// TIA Portal project "СrystallizerGorodenki" (V14)

(* hardware
DEVICE "ET 200SP station_1"  ET 200SP-Station
   slot 0: "Rack_0"  Rack  6ES5 710-8MAx1
   slot 1: "PLC_1"  CPU 1510SP-1 PN  6ES7 510-1DJ01-0AB0  V2.1
   slot 2: "AI 4xRTD/TC 2-,3-,4-wire HF_1"  AI 4xRTD/TC 2-,3-,4-wire HF  6ES7 134-6JD00-0CA1  V2.0
      slot 1: "AI 4xRTD/TC 2-,3-,4-wire HF_1"  AI 4xRTD/TC 2-,3-,4-wire HF
   slot 3: "AI 4xRTD/TC 2-,3-,4-wire HF_2"  AI 4xRTD/TC 2-,3-,4-wire HF  6ES7 134-6JD00-0CA1  V2.0
      slot 1: "AI 4xRTD/TC 2-,3-,4-wire HF_2"  AI 4xRTD/TC 2-,3-,4-wire HF
   slot 4: "AI 4xRTD/TC 2-,3-,4-wire HF_3"  AI 4xRTD/TC 2-,3-,4-wire HF  6ES7 134-6JD00-0CA1  V2.0
      slot 1: "AI 4xRTD/TC 2-,3-,4-wire HF_3"  AI 4xRTD/TC 2-,3-,4-wire HF
   slot 5: "AI 4xI 2-,4-wire ST_1"  AI 4xI 2-,4-wire ST  6ES7 134-6GD00-0BA1  V1.1
      slot 1: "AI 4xI 2-,4-wire ST_1"  AI 4xI 2-,4-wire ST
   slot 6: "AI 4xI 2-,4-wire ST_2"  AI 4xI 2-,4-wire ST  6ES7 134-6GD00-0BA1  V1.1
      slot 1: "AI 4xI 2-,4-wire ST_2"  AI 4xI 2-,4-wire ST
   slot 7: "DI 16x24VDC ST_1"  DI 16x24VDC ST  6ES7 131-6BH01-0BA0  V0.0
      slot 1: "DI 16x24VDC ST_1"  DI 16x24VDC ST
   slot 8: "DI 16x24VDC ST_2"  DI 16x24VDC ST  6ES7 131-6BH01-0BA0  V0.0
      slot 1: "DI 16x24VDC ST_2"  DI 16x24VDC ST
   slot 9: "DI 16x24VDC ST_3"  DI 16x24VDC ST  6ES7 131-6BH01-0BA0  V0.0
      slot 1: "DI 16x24VDC ST_3"  DI 16x24VDC ST
   slot 10: "DI 8x24VDC ST_1"  DI 8x24VDC ST  6ES7 131-6BF01-0BA0  V0.0
      slot 1: "DI 8x24VDC ST_1"  DI 8x24VDC ST
   slot 11: "DQ 16x24VDC/0.5A ST_1"  DQ 16x24VDC/0.5A ST  6ES7 132-6BH01-0BA0  V0.0
      slot 1: "DQ 16x24VDC/0.5A ST_1"  DQ 16x24VDC/0.5A ST
   slot 12: "DQ 8x24VDC/0.5A ST_1"  DQ 8x24VDC/0.5A ST  6ES7 132-6BF01-0BA0  V0.0
      slot 1: "DQ 8x24VDC/0.5A ST_1"  DQ 8x24VDC/0.5A ST
   slot 13: "AQ 2xI ST_1"  AQ 2xI ST  6ES7 135-6GB00-0BA1  V1.0
      slot 1: "AQ 2xI ST_1"  AQ 2xI ST
   slot 14: "Server module_1"  Server module  6ES7 193-6PA00-0AA0  V1.1
      slot 1: "Server module_1"  Server module
   slot 127: "BA 2xRJ45"  BA 2xRJ45  6ES7 193-6AR00-0AA0  V0.0
      slot 32769: "Port_1"  6ES7 193-6AR00-0AA0
      slot 32770: "Port_2"  6ES7 193-6AR00-0AA0
DEVICE "HMI_1"  TP900 Comfort
   slot 0: "TP900 Comfort"  TP900 Comfort  6AV2 124-0JC01-0AX0  14.0.1.0
   slot 1: "HMI_RT_1"  TP900 Comfort  6AV2 124-0JC01-0AX0  14.0.1.0
   slot 5: "HMI_1.IE_CP_1"  PROFINET Interface  14.0.1.0
      slot 1: "PROFINET Interface_1"  PROFINET Interface
         slot 1: "Port_1"  Port
         slot 2: "Port_2"  Port
   slot 7: "HMI_1.MPI/DP_CP_1"  MPI/DP Interface  14.0.1.0
DEVICE "GSD device_1"  GSD.Device.PN
   slot 0: "Rack"  Rack  V1.0
   slot 0: "CTEU-PN"  CTEU-PN  2201471  V1.0.0
      slot 0: "CTEU-PN"  CTEU-PN
      slot 1: "PN-IO Interface"  PN-IO Interface
         slot 1: "Port 1"  Port 1
         slot 2: "Port 2"  Port 2
   slot 1: "VAEM-L1-S-16-PT_1"  VAEM-L1-S-16-PT  573939
      slot 0: "VAEM-L1-S-16-PT"  VAEM-L1-S-16-PT
DEVICE "SINAMICS G_1"  Sinamics.Device
   slot 0: "	_0"  Rail
   slot 0: "M1_1"  G120C PN  6SL3210-1KE18-8UF1  4.7.6
      slot 3: "PM G120C"  PM G120C  6SL3210-1KE18-8UF1  -
DEVICE "SINAMICS G_2"  Sinamics.Device
   slot 0: "	_0"  Rail
   slot 0: "M2_1"  G120C PN  6SL3210-1KE18-8UF1  4.7.6
      slot 3: "PM G120C"  PM G120C  6SL3210-1KE18-8UF1  -
DEVICE "SINAMICS G_4"  Sinamics.Device
   slot 0: "	_0"  Rail
   slot 0: "M7_1"  G120C PN  6SL3210-1KE18-8UF1  4.7.6
      slot 3: "PM G120C"  PM G120C  6SL3210-1KE18-8UF1  -
DEVICE "SINAMICS G_5"  Sinamics.Device
   slot 0: "	_0"  Rail
   slot 0: "M7_2"  G120C PN  6SL3210-1KE21-3UF1  4.7.6
      slot 3: "PM G120C"  PM G120C  6SL3210-1KE21-3UF1  -
DEVICE "PC-System_1"  SIMATIC PC station
   slot 0: "PC station"  Rail  SIMATIC PC-Station  V1.0
      slot 125: "Stationmanager"  Station_Manager  V6.0.4
   slot 1: "IE general_1"  IE General  IE_CP  V8.2.0
   slot 2: "HMI_RT_3"  WinCC RT Advanced  6AV2 104-0xxxx-xxxx  14.0.1.0
      slot 33792: "Host interface"  Host interface
*)

// ===== PLC "PLC_1"  CPU 1510SP-1 PN =====

VAR_GLOBAL   // PLC tag table "Default tag table"
   "Ai_TE1.1" AT %IW0 : Int;
   "Ai_TE1.2" AT %IW2 : Int;
   "Ai_TE1.3" AT %IW4 : Int;
   "Ai_TE2.1" AT %IW6 : Int;
   "Ai_TE2.2" AT %IW8 : Int;
   "Ai_TE2.3" AT %IW10 : Int;
   "Ai_TE7.1" AT %IW12 : Int;
   "Ai_TE7.2" AT %IW14 : Int;
   "Ai_TE3.1" AT %IW16 : Int;
   "Ai_TE3.2" AT %IW18 : Int;
   "Ai_TE3.3" AT %IW20 : Int;
   "Ai_LIC1.1" AT %IW24 : Int;
   "Ai_LIC2.1" AT %IW28 : Int;
   "Ai_LIC7.1" AT %IW32 : Int;
   "Ai_LIC7.2" AT %IW38 : Int;
   "Di_KF01" AT %I40.0 : Bool;
   "Di_AvarStop" AT %I40.1 : Bool;
   "Di_ACK" AT %I40.2 : Bool;
   "Di_BatRaz" AT %I40.3 : Bool;
   "Di_BatFault" AT %I40.4 : Bool;
   "Di_Bat24Ok" AT %I40.5 : Bool;
   "Di_BatEnable" AT %I40.6 : Bool;
   "Di_Qf1.1" AT %I40.7 : Bool;
   "Di_Km1.2" AT %I41.0 : Bool;
   "Di_Qf2.1" AT %I41.1 : Bool;
   "Di_Km2.2" AT %I41.2 : Bool;
   "Di_Qf3.1" AT %I41.3 : Bool;
   "Di_Km3.2" AT %I41.4 : Bool;
   "Di_Km03" AT %I42.0 : Bool;
   "Di_Km04" AT %I42.1 : Bool;
   "Di_QF7.1" AT %I42.2 : Bool;
   "Di_QF7.2" AT %I42.3 : Bool;
   "Di_Km10" AT %I42.4 : Bool;
   "Di_Ksp01" AT %I42.5 : Bool;
   "Di_Lah1.1" AT %I42.6 : Bool;
   "Di_Lah2.1" AT %I42.7 : Bool;
   "Di_Lah3.1" AT %I43.0 : Bool;
   "Di_Lah01" AT %I43.1 : Bool;
   "Di_Lal01" AT %I43.2 : Bool;
   "Di_Ga1.1" AT %I44.0 : Bool;
   "Di_Ga1.2" AT %I44.1 : Bool;
   "Di_Ga1.3" AT %I44.2 : Bool;
   "Di_Ga1.4" AT %I44.3 : Bool;
   "Di_Ga2.1" AT %I44.4 : Bool;
   "Di_Ga2.2" AT %I44.5 : Bool;
   "Di_Ga2.3" AT %I44.6 : Bool;
   "Di_Ga2.4" AT %I44.7 : Bool;
   "Di_Ga3.1" AT %I45.0 : Bool;
   "Di_Ga3.2" AT %I45.1 : Bool;
   "Di_Ga3.3" AT %I45.2 : Bool;
   "Di_Ga3.4" AT %I45.3 : Bool;
   "Di_Ga7.3" AT %I45.4 : Bool;
   "Di_Ga7.4" AT %I45.5 : Bool;
   "Di_1Ga01" AT %I45.6 : Bool;
   "Di_1Ga02" AT %I46.0 : Bool;
   "Di_1Ga03" AT %I46.1 : Bool;
   "Di_1Ga04" AT %I46.2 : Bool;
   "Di_1Ga05" AT %I46.3 : Bool;
   "Di_1Ga06" AT %I46.4 : Bool;
   "Di_Ga1.7" AT %I46.5 : Bool;
   "Di_Ga2.7" AT %I46.6 : Bool;
   "Di_Ga3.7" AT %I46.7 : Bool;
   "Dq_KB1" AT %Q0.0 : Bool;
   "Dq_Km1.2" AT %Q0.1 : Bool;
   "Dq_Km2.2" AT %Q0.2 : Bool;
   "Dq_Km3.2" AT %Q0.3 : Bool;
   "Dq_Km3" AT %Q0.4 : Bool;
   "Dq_Km4" AT %Q0.5 : Bool;
   "Dq_Km10" AT %Q0.6 : Bool;
   "Dq_V7.1" AT %Q0.7 : Bool;
   "Dq_V7.2" AT %Q1.0 : Bool;
   "Dq_V1.1" AT %Q3.0 : Bool;
   "Dq_V2.1" AT %Q3.1 : Bool;
   "Dq_V3.1" AT %Q3.2 : Bool;
   "Dq_V1.7" AT %Q3.3 : Bool;
   "Dq_V2.7" AT %Q3.4 : Bool;
   "Dq_V3.7" AT %Q3.5 : Bool;
   "Dq_V7.3" AT %Q3.6 : Bool;
   "Dq_V7.4" AT %Q3.7 : Bool;
   "System_Byte" AT %MB0 : Byte;
   "_Start" AT %M0.0 : Bool;   // Первый цикл
   "DiagStatusUpdate" AT %M0.1 : Bool;
   "_T(1)" AT %M0.2 : Bool;   // Всегда TRUE
   "_F(0)" AT %M0.3 : Bool;   // Всегда FALSE
   "_Clock" AT %MB1 : Byte;   // Байт часов
   "_Clk01sec" AT %M1.0 : Bool;   // Период изменения бита - 0.1 сек
   "_Clk02sec" AT %M1.1 : Bool;   // Период изменения бита - 0.2 сек
   "_Clk04sec" AT %M1.2 : Bool;   // Период изменения бита - 0.4 сек
   "_Clk05sec" AT %M1.3 : Bool;   // Период изменения бита - 0.5 сек
   "_Clk08sec" AT %M1.4 : Bool;   // Период изменения бита - 0.8 сек
   "_Clk10sec" AT %M1.5 : Bool;   // Период изменения бита - 1.0 сек
   "_Clk16sec" AT %M1.6 : Bool;   // Период изменения бита - 1.6 сек
   "_Clk20sec" AT %M1.7 : Bool;   // Период изменения бита - 2.0 сек
   "_ReStart" AT %M2.0 : Bool;   // Выполняется первый проход OB1
   "_AiMd" AT %M2.1 : Bool;   // Принудительная настройка аналоговых каналов
   "_HALT" AT %M2.2 : Bool;   // Общий "Аварийный СТОП"
   "_ACK" AT %M2.3 : Bool;   // Общий "Квитирование"
   "_MEn" AT %M2.4 : Bool;   // Общее разрешение сообщений
   "_Time" AT %MD20 : Time;   // Текущее системное время
   "_Time_dR" AT %MD24 : Real;   // Время цикла
   "Ao_RV01" AT %QW7 : Int;
   "Tag_3" AT %M11.0 : Bool;
   "Tag_4" AT %M11.1 : Bool;
   "Tag_5" AT %M11.2 : Bool;
   "Tag_6" AT %M11.3 : Bool;
END_VAR

VAR_GLOBAL CONSTANT   // PLC tag table "Default tag table"
   "NLoo" : Real := -1.0e+38;   // Условный уровень -oo для показаний датчика
   "NHoo" : Real := 1.0e+38;   // Условный уровень +oo для показаний датчика
   "TS0" : LDT := LDT#1970-01-01-00:00:00;   // Program_Alarm.TIMESTAMP := #TS0
   "Tz" : Time := T#0ms;   // Инициализация переменных времени
END_VAR

TYPE "PID"
   STRUCT
      Man_On : Bool;
      Man : Real;
      Sp : Real;
      LMN : Real;
   END_STRUCT;
END_TYPE

// folder: _LIB

TYPE "DrvST"
TITLE = 'Структура слова командного канала DrvCell побайтно'
VERSION : 0.1
   STRUCT
      STx : Byte := 16#00;   // [0_] Статус механизма
      WKx : Byte := 16#00;   // [1_] Вспомогательные данные канала
      Cmd : Byte := 16#00;   // [2_] Текущая команда и штамп идентификатора команды
      SPx : SInt := 0;   // [3_] Текущая уставка (-100..+100)[%]
   END_STRUCT;
END_TYPE

TYPE "DrvCF"
TITLE = 'Структура слова командного канала DrvCell побитно'
VERSION : 0.1
   STRUCT
      Sx1 : Bool := 0;   // [00] SQ канала Km1
      Sx2 : Bool := 0;   // [01] SQ канала Km2
      Ks1 : Bool := 0;   // [02] Включен канал Km1
      Ks2 : Bool := 0;   // [03] Включен канал Km2
      Tm1 : Bool := 0;   // [04] Время Tm1 истекло
      Tm2 : Bool := 0;   // [05] Время Tm2 истекло
      Er1 : Bool := 0;   // [06] Неисправность Km1
      Er2 : Bool := 0;   // [07] Неисправность Km2
      Act : Bool := 0;   // [10] Актуальность данных (контроль обрыва связи)
      Ack : Bool := 0;   // [11] Квитирование ошибок
      MsD : Bool := 0;   // [12] Сообщение: Наличие обрыва связи
      MsB : Bool := 0;   // [13] Сообщение: Наличие блокировки команды
      Mdx : Bool := 0;   // [14] Режим работы DrvCell (0==Ручной/1==Автомат)
      F15 : Bool := 0;   // [15] Резерв
      F16 : Bool := 0;   // [16] Резерв
      F17 : Bool := 0;   // [17] Резерв
      Cm0 : Bool := 0;   // [20] Команда: бит 0
      Cm1 : Bool := 0;   // [21] Команда: бит 1
      Cm2 : Bool := 0;   // [22] Команда: бит 2
      F23 : Bool := 0;   // [23] Резерв
      F24 : Bool := 0;   // [24] Резерв
      F25 : Bool := 0;   // [25] Резерв
      F26 : Bool := 0;   // [26] Резерв
      F27 : Bool := 0;   // [27] Резерв
      SPx : SInt := 0;   // [3_] Текущая уставка (-100..+100)[%]
   END_STRUCT;
END_TYPE

TYPE "DrvNm"
TITLE = 'Данные канала системы блокировок'
VERSION : 0.1
   STRUCT
      Ds1 : Bool := 0;   // Блокировка включения (принудительное отключение) Km1
      Ds2 : Bool := 0;   // Блокировка включения (принудительное отключение) Km2
      DsA : Bool := 0;   // Общая блокировка включения (принудительное отключение) Km1&Km2
      r03 : Bool := 0;   // ----
      r04 : Bool := 0;   // ----
      r05 : Bool := 0;   // ----
      r06 : Bool := 0;   // ----
      r07 : Bool := 0;   // ----
      MsA : Byte := 16#00;   // Номер сообщения общей блокировки
      Ms2 : Byte := 16#00;   // Номер сообщения блокировки включения Km2
      Ms1 : Byte := 16#00;   // Номер сообщения блокировки включения Km1
   END_STRUCT;
END_TYPE

TYPE "DrvMs"
TITLE = 'Расшифровка слова состояния HMI DrvCell побитно'
VERSION : 0.1
   STRUCT
      Ds1 : Bool := 0;   // Действие Km1 заблокировано (Ds1/DsA)
      Ds2 : Bool := 0;   // Действие Km2 заблокировано (Ds2/DsA)
      QFe : Bool := 0;   // Отключен автоматический выключатель
      Flt : Bool := 0;   // Внешняя неисправность (блокирующая)
      Err : Bool := 0;   // Внутренняя неисправность DrvCell
      b29 : Bool := 0;   // ----
      b30 : Bool := 0;   // ----
      b31 : Bool := 0;   // ----
      Sr1 : Bool := 0;   // Не сработал КВ SQ1 за заданное время Tm1
      Sr2 : Bool := 0;   // Не сработал КВ SQ2 за заданное время Tm2
      Se1 : Bool := 0;   // Механиз без команды сошел с КВ SQ1
      Se2 : Bool := 0;   // Механиз без команды сошел с КВ SQ2
      SeA : Bool := 0;   // Одновременно активны оба КВ SQ1 и SQ2
      KeB : Bool := 0;   // БК KxB не соответствует состоянию KOn
      Ke1 : Bool := 0;   // БК Kx1 не соответствует контактору Km1
      Ke2 : Bool := 0;   // БК Kx2 не соответствует контактору Km2
      Mdx : Bool := 0;   // Режим работы DrvCell (0==Ручной/1==Автомат)
      Lg2 : Bool := 0;   // Индикация действия от SB2 (зеленый)
      Ly2 : Bool := 0;   // Индикация действия от SB2 (желтый)
      Lr2 : Bool := 0;   // Индикация действия от SB2 (красный)
      HSB : Bool := 0;   // Доп. признак индикации SB2
      Lg1 : Bool := 0;   // Индикация действия от SB1 (зеленый)
      Ly1 : Bool := 0;   // Индикация действия от SB1 (желтый)
      Lr1 : Bool := 0;   // Индикация действия от SB1 (красный)
      Sx1 : Bool := 0;   // Активное состояние SQ1
      Sx2 : Bool := 0;   // Активное состояние SQ2
      Ks1 : Bool := 0;   // Запрос на включение Km1
      Ks2 : Bool := 0;   // Запрос на включение Km2
      Tm1 : Bool := 0;   // Время Tm1 истекло
      Tm2 : Bool := 0;   // Время Tm2 истекло
      Er1 : Bool := 0;   // Неисправность Km1
      Er2 : Bool := 0;   // Неисправность Km2
   END_STRUCT;
END_TYPE

TYPE "TPTR"
TITLE = 'Формат данных типа POINTER'
VERSION : 0.1
   STRUCT
      DN : UInt := 0;   // DB number
      AR : UDInt := 0;   // Memory area
   END_STRUCT;
END_TYPE

TYPE "TANY"
TITLE = 'Формат данных типа ANY'
VERSION : 0.1
   STRUCT
      S7 : Byte := B#16#00;   // 10h for S7
      TP : Byte := B#16#00;   // Data type
      RF : UInt := 0;   // Repetition factor
      PTR : "TPTR";   // POINTER
   END_STRUCT;
END_TYPE

TYPE "AiSP"
TITLE = 'Параметры настройки входного аналогового канала'
VERSION : 0.1
   STRUCT
      "M" : Struct   // Общая мастер-структура параметров каналов
         Rz : Bool := 1;   // При Rz<>Rs производится перерасчет канала
         Rs : Bool := 0;   // По фронту изменения Rs производится перенастройка канала
         Nm : Bool := 0;   // Pn указывает нормальный==0/номинальный==1 сигнал
         Ke : Bool := 0;   // Прямое использование Kf и Zp (с перерассчетом P1 и P0)
         Ms : Bool := 1;   // Разрешена генерация сообщений и использование Pn
         Rt : Bool := 0;   // Круговой датчик с переходом через 0 (однооборотный/многооборотный)
         Rh : Bool := 1;   // Для кругового датчика использовать шкалу со знаком (-180*..+180*)
         R0 : Word := 16#0000;   // ----
         An : DInt := DINT#27648;   // Значение PIW/PID(Ai/Ad) при 100% входного диапазона
         P1 : Real := 100.0;   // Номинал Px при Ai=100% (Ai=An[1]) [E]
         P0 : Real := 0.0;   // Номинал Px при Ai=0% (Ai=0[1]) [E]
         Kf : Real := 1.0;   // Коэффициент преобразования Ai=>Px (множитель) [E/1]
         Kx : Real := 1.0;   // Множитель для сглаживания колебаний входного сигнала
         dP : Real := 0.0;   // Гистерезис в определении уровней
      END_STRUCT;
      Pn : Real := 1.0e+38;   // Номинальный/Нормальный уровень сигнала [E]
      Ha : Real := 1.0e+38;   // Верхний уровень сигнала: Аварийный [E/%]
      La : Real := -1.0e+38;   // Нижний уровень сигнала: Аварийный [E/%]
      Hw : Real := 1.0e+38;   // Верхний уровень сигнала: Предупредительный [E/%]
      Lw : Real := -1.0e+38;   // Нижний уровень сигнала: Предупредительный [E/%]
      H1 : Real := 1.0e+38;   // Верхний уровень сигнала: Рабочая зона 1 [E/%]
      L1 : Real := -1.0e+38;   // Нижний уровень сигнала: Рабочая зона 1 [E/%]
      H0 : Real := 1.0e+38;   // Верхний уровень сигнала: Рабочая зона 0 [E/%]
      L0 : Real := -1.0e+38;   // Нижний уровень сигнала: Рабочая зона 0 [E/%]
   END_STRUCT;
END_TYPE

TYPE "DrvRd"
TITLE = 'Данные канала резервирования приводов'
VERSION : 0.1
   STRUCT
      S : Struct
         Mst : Bool := 1;   // Данный привод является основным (Master==1/Slave==0)
         Rd1 : Bool := 1;   // Данный привод включен как основной
         Rd2 : Bool := 0;   // Данный привод включен как резервный
         Dis : Bool := 0;   // Запрет использования привода (блокировка)
         r0 : Word := 16#0000;   // ---- Структура статуса (состояния) резерва
      END_STRUCT;
      "M" : Struct
         UBr : Bool := 0;   // Безусловное растормаживание (расжать)
         Enb : Bool := 0;   // Разрешение работы (разблокирование)
         KOn : Bool := 0;   // Включить намагничивание V=0 (команда)
         Run : Bool := 0;   // Пуск привода V=Vs (команда)
         Ack : Bool := 0;   // Сброс индикации ошибки (квитирование) (1==активен)
         Id : Word := 16#0000;   // Идентификатор дополнительных параметров привода
         Ms : Real := 0.0;   // Заданный момент [%]
         Vs : Real := 0.0;   // Заданная скорость [E]
         Vn : Real := 100.0;   // Номинальная скорость [E] Структура параметров мастера резерва
      END_STRUCT;
      X : Struct
         Brk : Bool := 0;   // Привод включен (разблокировка тормоза).
         Err : Bool := 0;   // Неисправность/авария привода
         Rdy : Bool := 0;   // Готовность привода к включению
         SW : Word := 16#0000;   // Текущее слово состояния привода
         Vx : Real := 0.0;   // Текущая скорость привода [E]
         Ix : Real := 0.0;   // Текущий ток привода [%]
         Mx : Real := 0.0;   // Текущий момент привода [%]
         An : Int := 0;   // Текущий номер сигнала Alarm [№] (предупреждение) (либо альтернативные данные)
         Fn : Int := 0;   // Текущий номер сигнала Fault [№] (отказ) Структура состояния привода
      END_STRUCT;
   END_STRUCT;
END_TYPE

TYPE "DrvME"
VERSION : 0.1
   STRUCT
      Pr : Struct   // Структура параметров сообщения ALARM
         N1 : UDInt := 0;   // Именная строка сообщения (MSGS=GRP)
         N2 : UDInt := 0;   // Признаки состояния сообщения (MSGS=MEn/Mdx/KOn)
         N3 : UDInt := 0;   // Основное сообщение (MSGS=A)
         N4 : UDInt := 0;   // Вспомогательное сообщение (MSGS=B)
         N5 : UDInt := 0;   // Вспомогательное сообщение (MSGS=C)
         N6 : UDInt := 0;   // Дополнительная строка сообщения (MSGS=GRP+N)
      END_STRUCT;
   END_STRUCT;
END_TYPE

TYPE "AiSF"
VERSION : 0.1
   STRUCT
      b24 : Bool;   // ----
      b25 : Bool;   // ----
      b26 : Bool;   // ----
      b27 : Bool;   // ----
      MEn : Bool;   // Разрешение выдачи сообщений (HMI)
      b29 : Bool;   // ----
      b30 : Bool;   // ----
      QSt : Bool;   // Настройка блока выполнена
      LSP : Bool;   // Запрос установки смещения (PLC)
      HSP : Bool;   // Запрос установки смещения (HMI)
      ESP : Bool;   // Разрешение установки смещения (HMI)
      QSP : Bool;   // Признак установки смещения
      LFQ : Bool;   // Запрос режима форсирования (PLC)
      HFQ : Bool;   // Запрос режима форсирования (HMI)
      EFQ : Bool;   // Разрешение режима форсирования (HMI)
      QFQ : Bool;   // Признак режима форсирования
      QWg : Bool;   // Наличие предупреждения
      QAm : Bool;   // Наличие аварии
      QFt : Bool;   // Наличие неисправности канала
      b11 : Bool;   // ----
      b12 : Bool;   // ----
      b13 : Bool;   // ----
      HWg : Bool;   // Наличие предупреждения (HMI:Yellow)
      HAm : Bool;   // Наличие аварии/неисправности (HMI:Red)
      QL0 : Bool;   // Нижний уровень сигнала: Рабочая зона 0
      QH0 : Bool;   // Верхний уровень сигнала: Рабочая зона 0
      QL1 : Bool;   // Нижний уровень сигнала: Рабочая зона 1
      QH1 : Bool;   // Верхний уровень сигнала: Рабочая зона 1
      QLw : Bool;   // Нижний уровень сигнала: Предупредительный
      QHw : Bool;   // Верхний уровень сигнала: Предупредительный
      QLa : Bool;   // Нижний уровень сигнала: Аварийный
      QHa : Bool;   // Верхний уровень сигнала: Аварийный
   END_STRUCT;
END_TYPE

// folder: Ai

DATA_BLOCK "AiCh_TE1.1"   // DB1
{ S7_Optimized_Access := 'FALSE' }
VERSION : 0.1
// stored: InstanceOfName AiCh_My
"AiCh_My"
BEGIN
END_DATA_BLOCK

DATA_BLOCK "AiCh_TE1.2"   // DB2
{ S7_Optimized_Access := 'FALSE' }
VERSION : 0.1
// stored: InstanceOfName AiCh_My
"AiCh_My"
BEGIN
END_DATA_BLOCK

DATA_BLOCK "AiCh_TE1.3"   // DB3
{ S7_Optimized_Access := 'FALSE' }
VERSION : 0.1
// stored: InstanceOfName AiCh_My
"AiCh_My"
BEGIN
END_DATA_BLOCK

DATA_BLOCK "AiCh_TE2.1"   // DB4
{ S7_Optimized_Access := 'FALSE' }
VERSION : 0.1
// stored: InstanceOfName AiCh_My
"AiCh_My"
BEGIN
END_DATA_BLOCK

DATA_BLOCK "AiCh_TE2.2"   // DB5
{ S7_Optimized_Access := 'FALSE' }
VERSION : 0.1
// stored: InstanceOfName AiCh_My
"AiCh_My"
BEGIN
END_DATA_BLOCK

DATA_BLOCK "AiCh_TE2.3"   // DB6
{ S7_Optimized_Access := 'FALSE' }
VERSION : 0.1
// stored: InstanceOfName AiCh_My
"AiCh_My"
BEGIN
END_DATA_BLOCK

DATA_BLOCK "AiCh_TE7.1"   // DB7
{ S7_Optimized_Access := 'FALSE' }
VERSION : 0.1
// stored: InstanceOfName AiCh_My
"AiCh_My"
BEGIN
END_DATA_BLOCK

DATA_BLOCK "AiCh_TE7.2"   // DB8
{ S7_Optimized_Access := 'FALSE' }
VERSION : 0.1
// stored: InstanceOfName AiCh_My
"AiCh_My"
BEGIN
END_DATA_BLOCK

DATA_BLOCK "AiCh_TE3.1"   // DB9
{ S7_Optimized_Access := 'FALSE' }
VERSION : 0.1
// stored: InstanceOfName AiCh_My
"AiCh_My"
BEGIN
END_DATA_BLOCK

DATA_BLOCK "AiCh_TE3.2"   // DB10
{ S7_Optimized_Access := 'FALSE' }
VERSION : 0.1
// stored: InstanceOfName AiCh_My
"AiCh_My"
BEGIN
END_DATA_BLOCK

DATA_BLOCK "AiCh_TE3.3"   // DB11
{ S7_Optimized_Access := 'FALSE' }
VERSION : 0.1
// stored: InstanceOfName AiCh_My
"AiCh_My"
BEGIN
END_DATA_BLOCK

DATA_BLOCK "AiCh_LIC1.1"   // DB12
{ S7_Optimized_Access := 'FALSE' }
VERSION : 0.1
// stored: InstanceOfName AiCh_My
"AiCh_My"
BEGIN
END_DATA_BLOCK

DATA_BLOCK "AiCh_LIC2.1"   // DB13
{ S7_Optimized_Access := 'FALSE' }
VERSION : 0.1
// stored: InstanceOfName AiCh_My
"AiCh_My"
BEGIN
END_DATA_BLOCK

DATA_BLOCK "AiCh_LIC3.1"   // DB14
{ S7_Optimized_Access := 'FALSE' }
VERSION : 0.1
// stored: InstanceOfName AiCh_My
"AiCh_My"
BEGIN
END_DATA_BLOCK

DATA_BLOCK "AiCh_LIC7.1"   // DB15
{ S7_Optimized_Access := 'FALSE' }
VERSION : 0.1
// stored: InstanceOfName AiCh_My
"AiCh_My"
BEGIN
END_DATA_BLOCK

DATA_BLOCK "AiCh_LIC7.2"   // DB16
{ S7_Optimized_Access := 'FALSE' }
VERSION : 0.1
// stored: InstanceOfName AiCh_My
"AiCh_My"
BEGIN
END_DATA_BLOCK

DATA_BLOCK "ForVO_DB"   // DB60
{ S7_Optimized_Access := 'FALSE' }
VERSION : 0.1
// stored: InstanceOfName ForVO
"ForVO"
BEGIN
END_DATA_BLOCK

// folder: Drives

DATA_BLOCK "DriveM1_1"   // DB33
{ S7_Optimized_Access := 'FALSE' }
AUTHOR : AA
FAMILY : xDEVICE
VERSION : 0.1
// stored: InstanceOfName MM_T352
"MM_T352"
BEGIN
END_DATA_BLOCK

DATA_BLOCK "DriveM7_1"   // DB34
{ S7_Optimized_Access := 'FALSE' }
AUTHOR : AA
FAMILY : xDEVICE
VERSION : 0.1
// stored: InstanceOfName MM_T352
"MM_T352"
BEGIN
END_DATA_BLOCK

DATA_BLOCK "DriveM7_2"   // DB35
{ S7_Optimized_Access := 'FALSE' }
AUTHOR : AA
FAMILY : xDEVICE
VERSION : 0.1
// stored: InstanceOfName MM_T352
"MM_T352"
BEGIN
END_DATA_BLOCK

DATA_BLOCK "DriveM2_1"   // DB38
{ S7_Optimized_Access := 'FALSE' }
AUTHOR : AA
FAMILY : xDEVICE
VERSION : 0.1
// stored: InstanceOfName MM_T352
"MM_T352"
BEGIN
END_DATA_BLOCK

// folder: Errors

DATA_BLOCK "FpDW_DB"   // DB43
{ S7_Optimized_Access := 'FALSE' }
VERSION : 0.1
// stored: InstanceOfName FpDW
"FpDW"
BEGIN
END_DATA_BLOCK

// folder: IceWater

DATA_BLOCK "IceWaterWork_DB"   // DB61
{ S7_Optimized_Access := 'TRUE' }
VERSION : 0.1
// stored: InstanceOfName IceWaterWork
"IceWaterWork"
BEGIN
END_DATA_BLOCK

// folder: KristalizersWork

DATA_BLOCK "Kr_2_Work"   // DB45
{ S7_Optimized_Access := 'TRUE' }
VERSION : 0.1
// stored: InstanceOfName KristalizerWork
"KristalizerWork"
BEGIN
END_DATA_BLOCK

DATA_BLOCK "Mixer2_Work_DB"   // DB47
{ S7_Optimized_Access := 'TRUE' }
VERSION : 0.1
// stored: InstanceOfName MixerWork
"MixerWork"
BEGIN
END_DATA_BLOCK

DATA_BLOCK "Mixer1_Work_DB"   // DB48
{ S7_Optimized_Access := 'TRUE' }
VERSION : 0.1
// stored: InstanceOfName MixerWork
"MixerWork"
BEGIN
END_DATA_BLOCK

DATA_BLOCK "Kr_1_Work"   // DB63
{ S7_Optimized_Access := 'TRUE' }
VERSION : 0.1
// stored: InstanceOfName KristalizerWork
"KristalizerWork"
BEGIN
END_DATA_BLOCK

// folder: Lines

DATA_BLOCK "ViewLine_DB"   // DB58
{ S7_Optimized_Access := 'TRUE' }
VERSION : 0.1
// stored: InstanceOfName ViewLine
"ViewLine"
BEGIN
END_DATA_BLOCK

// folder: Messages

DATA_BLOCK "Messages"   // DB44
{ S7_Optimized_Access := 'FALSE' }
VERSION : 0.1
   VAR
      Message1 : Bool;
      Message2 : Bool;
      Message3 : Bool;
      Message4 : Bool;
      Message5 : Bool;
      Message6 : Bool;
      Message7 : Bool;
      Message8 : Bool;
      Message9 : Bool;
      Message10 : Bool;
      Message11 : Bool;
      Message12 : Bool;
      Message13 : Bool;
      Message14 : Bool;
      Message15 : Bool;
      Message16 : Bool;
   END_VAR
BEGIN
END_DATA_BLOCK

// folder: Pumps&Valves

DATA_BLOCK "DrvCell_M1_2"   // DB17
{ S7_Optimized_Access := 'FALSE' }
AUTHOR : SAA
FAMILY : xDRIVER
NAME : DrvCell
VERSION : 4.0
// stored: InstanceOfName DrvCell
"DrvCell"
BEGIN
END_DATA_BLOCK

DATA_BLOCK "DrvCell_M2_2"   // DB18
{ S7_Optimized_Access := 'FALSE' }
AUTHOR : SAA
FAMILY : xDRIVER
NAME : DrvCell
VERSION : 4.0
// stored: InstanceOfName DrvCell
"DrvCell"
BEGIN
END_DATA_BLOCK

DATA_BLOCK "DrvCell_M3_2"   // DB19
{ S7_Optimized_Access := 'FALSE' }
AUTHOR : SAA
FAMILY : xDRIVER
NAME : DrvCell
VERSION : 4.0
// stored: InstanceOfName DrvCell
"DrvCell"
BEGIN
END_DATA_BLOCK

DATA_BLOCK "DrvCell_M3"   // DB20
{ S7_Optimized_Access := 'FALSE' }
AUTHOR : SAA
FAMILY : xDRIVER
NAME : DrvCell
VERSION : 4.0
// stored: InstanceOfName DrvCell
"DrvCell"
BEGIN
END_DATA_BLOCK

DATA_BLOCK "DrvCell_M4"   // DB21
{ S7_Optimized_Access := 'FALSE' }
AUTHOR : SAA
FAMILY : xDRIVER
NAME : DrvCell
VERSION : 4.0
// stored: InstanceOfName DrvCell
"DrvCell"
BEGIN
END_DATA_BLOCK

DATA_BLOCK "DrvCell_M10"   // DB22
{ S7_Optimized_Access := 'FALSE' }
AUTHOR : SAA
FAMILY : xDRIVER
NAME : DrvCell
VERSION : 4.0
// stored: InstanceOfName DrvCell
"DrvCell"
BEGIN
END_DATA_BLOCK

DATA_BLOCK "DrvCell_V7_1"   // DB23
{ S7_Optimized_Access := 'FALSE' }
AUTHOR : SAA
FAMILY : xDRIVER
NAME : DrvCell
VERSION : 4.0
// stored: InstanceOfName DrvCell
"DrvCell"
BEGIN
END_DATA_BLOCK

DATA_BLOCK "DrvCell_V7_2"   // DB24
{ S7_Optimized_Access := 'FALSE' }
AUTHOR : SAA
FAMILY : xDRIVER
NAME : DrvCell
VERSION : 4.0
// stored: InstanceOfName DrvCell
"DrvCell"
BEGIN
END_DATA_BLOCK

DATA_BLOCK "DrvCell_V1_1"   // DB25
{ S7_Optimized_Access := 'FALSE' }
AUTHOR : SAA
FAMILY : xDRIVER
NAME : DrvCell
VERSION : 4.0
// stored: InstanceOfName DrvCell
"DrvCell"
BEGIN
END_DATA_BLOCK

DATA_BLOCK "DrvCell_V2_1"   // DB26
{ S7_Optimized_Access := 'FALSE' }
AUTHOR : SAA
FAMILY : xDRIVER
NAME : DrvCell
VERSION : 4.0
// stored: InstanceOfName DrvCell
"DrvCell"
BEGIN
END_DATA_BLOCK

DATA_BLOCK "DrvCell_V3_1"   // DB27
{ S7_Optimized_Access := 'FALSE' }
AUTHOR : SAA
FAMILY : xDRIVER
NAME : DrvCell
VERSION : 4.0
// stored: InstanceOfName DrvCell
"DrvCell"
BEGIN
END_DATA_BLOCK

DATA_BLOCK "DrvCell_V1_7"   // DB28
{ S7_Optimized_Access := 'FALSE' }
AUTHOR : SAA
FAMILY : xDRIVER
NAME : DrvCell
VERSION : 4.0
// stored: InstanceOfName DrvCell
"DrvCell"
BEGIN
END_DATA_BLOCK

DATA_BLOCK "DrvCell_V2_7"   // DB29
{ S7_Optimized_Access := 'FALSE' }
AUTHOR : SAA
FAMILY : xDRIVER
NAME : DrvCell
VERSION : 4.0
// stored: InstanceOfName DrvCell
"DrvCell"
BEGIN
END_DATA_BLOCK

DATA_BLOCK "DrvCell_V3_7"   // DB30
{ S7_Optimized_Access := 'FALSE' }
AUTHOR : SAA
FAMILY : xDRIVER
NAME : DrvCell
VERSION : 4.0
// stored: InstanceOfName DrvCell
"DrvCell"
BEGIN
END_DATA_BLOCK

DATA_BLOCK "DrvCell_V7_3"   // DB31
{ S7_Optimized_Access := 'FALSE' }
AUTHOR : SAA
FAMILY : xDRIVER
NAME : DrvCell
VERSION : 4.0
// stored: InstanceOfName DrvCell
"DrvCell"
BEGIN
END_DATA_BLOCK

DATA_BLOCK "DrvCell_V7_4"   // DB32
{ S7_Optimized_Access := 'FALSE' }
AUTHOR : SAA
FAMILY : xDRIVER
NAME : DrvCell
VERSION : 4.0
// stored: InstanceOfName DrvCell
"DrvCell"
BEGIN
END_DATA_BLOCK

DATA_BLOCK "DrvCell_M1_1"   // DB36
{ S7_Optimized_Access := 'FALSE' }
AUTHOR : SAA
FAMILY : xDRIVER
NAME : DrvCell
VERSION : 4.0
// stored: InstanceOfName DrvCell
"DrvCell"
BEGIN
END_DATA_BLOCK

DATA_BLOCK "DrvCell_M2_1"   // DB37
{ S7_Optimized_Access := 'FALSE' }
AUTHOR : SAA
FAMILY : xDRIVER
NAME : DrvCell
VERSION : 4.0
// stored: InstanceOfName DrvCell
"DrvCell"
BEGIN
END_DATA_BLOCK

DATA_BLOCK "DrvCell_M7_1"   // DB39
{ S7_Optimized_Access := 'FALSE' }
AUTHOR : SAA
FAMILY : xDRIVER
NAME : DrvCell
VERSION : 4.0
// stored: InstanceOfName DrvCell
"DrvCell"
BEGIN
END_DATA_BLOCK

DATA_BLOCK "DrvCell_M7_2"   // DB40
{ S7_Optimized_Access := 'FALSE' }
AUTHOR : SAA
FAMILY : xDRIVER
NAME : DrvCell
VERSION : 4.0
// stored: InstanceOfName DrvCell
"DrvCell"
BEGIN
END_DATA_BLOCK

DATA_BLOCK "DrvCell_M5"   // DB59
{ S7_Optimized_Access := 'FALSE' }
AUTHOR : SAA
FAMILY : xDRIVER
NAME : DrvCell
VERSION : 4.0
// stored: InstanceOfName DrvCell
"DrvCell"
BEGIN
END_DATA_BLOCK

// folder: Share

DATA_BLOCK "Data"   // DB41
{ S7_Optimized_Access := 'TRUE' }
VERSION : 0.1
   VAR
      Ack : Bool;
      GlobalError : Bool;
      GlobalErrorStop : Bool;
   END_VAR
   VAR RETAIN
      Reg_01RV01 : "PID";
      Reg_M7_1 : "PID";
   END_VAR
   VAR
      Reg_M7_2 : "PID";
      Reg_TE1_1 : Struct
         In : Bool := FALSE;
         Sp : Real := 0.0;
         Gis : Real := 0.1;
         V1_1 : Bool := FALSE;
      END_STRUCT;
      Reg_TE2_1 : Struct
         In : Bool := FALSE;
         Sp : Real := 0.0;
         Gis : Real := 0.1;
         V2_1 : Bool := FALSE;
      END_STRUCT;
   END_VAR
   VAR RETAIN
      Mixer1 : Struct
         Man : Real;
         Start : Bool;
         Stop : Bool;
         RegimBothSide : Bool := true;
         Power : Real := 50.0;
         TimeRight : DInt := 60;
         TimeLeft : DInt := 60;
         TimePause : DInt := 60;
         Direction : Int;
      END_STRUCT;
      Mixer2 : Struct
         Man : Real;
         Start : Bool;
         Stop : Bool;
         RegimBothSide : Bool := true;
         Power : Real := 50.0;
         TimeRight : DInt := 60;
         TimeLeft : DInt := 60;
         TimePause : DInt := 60;
         Direction : Int;
      END_STRUCT;
   END_VAR
   VAR
      MAN_ON : Bool;
      washing : Struct
         cipRegim : Int := 1;
         readyGlobal : Bool;
         readyRoute : Bool;
         Start : Bool;
         Stop : Bool;
      END_STRUCT;
      LevelVO_Pv : Real;
   END_VAR
   VAR RETAIN
      TempIn_Sp : Real := 30.0;
      Power_7_2 : Real := 40.0;
      Power_7_2_CIP : Real := 40.0;
   END_VAR
   VAR
      Kr1 : Struct
         Regim : Int := 1;
         TempFilling : Real := 30.0;
         TempKristal : Real := 15.0;
         TimeKristal : Int := 8;
         Start : Bool;
         Stop : Bool;
         Ready_Route : Bool;
         Ready_Work : Bool;
         Kr1 : Struct
            Regim : Int := 1;
            TempFilling : Real := 30.0;
            TempKristal : Real := 15.0;
            TimeKristal : Int := 8;
            Start : Bool;
            Stop : Bool;
            Ready_Route : Bool;
            Ready_Work : Bool;
         END_STRUCT;
      END_STRUCT;
      Kr2 : Struct
         Regim : Int := 1;
         TempFilling : Real := 30.0;
         TempKristal : Real := 15.0;
         TimeKristal : Int := 8;
         Start : Bool;
         Stop : Bool;
         Ready_Route : Bool;
         Ready_Work : Bool;
      END_STRUCT;
      TE1_1_SP : Real;
      Mixer1_Run : Bool;
      Mixer2_Run : Bool;
      Front_Mixer_1 : Bool;
      Front_Mixer_2 : Bool;
      Erorrs_Beep : Bool;
      KR1_Beep : Bool;
      KR2_Beep : Bool;
      Equipment_Work : Bool;
      ReadyCIP : Bool;
      ReadyKr1 : Bool;
      ReadyKr2 : Bool;
   END_VAR
   VAR RETAIN
      EnableReady : Bool := true;
   END_VAR
BEGIN
   Reg_M7_1.Sp := 10.0;
   Reg_01RV01.Sp := 30.0;
END_DATA_BLOCK

// folder: Sys

DATA_BLOCK "Sys_DB"   // DB42
{ S7_Optimized_Access := 'TRUE' }
VERSION : 0.1
// stored: InstanceOfName Sys
"Sys"
BEGIN
END_DATA_BLOCK

DATA_BLOCK "Panel_AreaPointer"   // DB105
{ S7_Optimized_Access := 'FALSE' }
VERSION : 0.1
   VAR
      Coordination : Word;
      DateTime : Date_And_Time;
      JobMailbox : Array[0..3] of Word;
      DataRecord : Array[0..4] of Word;
      ProjectID : Word;
      ScreenNumber : Array[0..4] of Word;
      DateTimePLC : Struct
         DateTime : Date_And_Time;
         Reserve_01 : Word;
         Reserve_02 : Word;
      END_STRUCT;
   END_VAR
BEGIN
END_DATA_BLOCK

// folder: System blocks/Program resources

DATA_BLOCK "IEC_Timer_0_DB"   // DB52
{ S7_Optimized_Access := 'TRUE' }
AUTHOR : Simatic
FAMILY : IEC
NAME : IEC_TMR
VERSION : 1.0
// stored: InstanceOfName IEC_TIMER
"IEC_TIMER"
BEGIN
END_DATA_BLOCK

DATA_BLOCK "IEC_Timer_0_DB_1"   // DB53
{ S7_Optimized_Access := 'TRUE' }
AUTHOR : Simatic
FAMILY : IEC
NAME : IEC_TMR
VERSION : 1.0
// stored: InstanceOfName IEC_TIMER
"IEC_TIMER"
BEGIN
END_DATA_BLOCK

DATA_BLOCK "IEC_Timer_0_DB_2"   // DB54
{ S7_Optimized_Access := 'TRUE' }
AUTHOR : Simatic
FAMILY : IEC
NAME : IEC_TMR
VERSION : 1.0
// stored: InstanceOfName IEC_TIMER
"IEC_TIMER"
BEGIN
END_DATA_BLOCK

DATA_BLOCK "IEC_Timer_0_DB_4"   // DB55
{ S7_Optimized_Access := 'TRUE' }
AUTHOR : Simatic
FAMILY : IEC
NAME : IEC_TMR
VERSION : 1.0
// stored: InstanceOfName IEC_TIMER
"IEC_TIMER"
BEGIN
END_DATA_BLOCK

DATA_BLOCK "IEC_Timer_0_DB_5"   // DB56
{ S7_Optimized_Access := 'TRUE' }
AUTHOR : Simatic
FAMILY : IEC
NAME : IEC_TMR
VERSION : 1.0
// stored: InstanceOfName IEC_TIMER
"IEC_TIMER"
BEGIN
END_DATA_BLOCK

DATA_BLOCK "IEC_Timer_0_DB_6"   // DB57
{ S7_Optimized_Access := 'TRUE' }
AUTHOR : Simatic
FAMILY : IEC
NAME : IEC_TMR
VERSION : 1.0
// stored: InstanceOfName IEC_TIMER
"IEC_TIMER"
BEGIN
END_DATA_BLOCK

DATA_BLOCK "IEC_Timer_0_DB_3"   // DB62
{ S7_Optimized_Access := 'TRUE' }
AUTHOR : Simatic
FAMILY : IEC
NAME : IEC_TMR
VERSION : 1.0
// stored: InstanceOfName IEC_TIMER
"IEC_TIMER"
BEGIN
END_DATA_BLOCK

// folder: Washing

DATA_BLOCK "WashingWork_DB"   // DB49
{ S7_Optimized_Access := 'TRUE' }
VERSION : 0.1
// stored: InstanceOfName WashingWork
"WashingWork"
BEGIN
END_DATA_BLOCK

// folder: (top level)

ORGANIZATION_BLOCK "Main"   // OB1, LAD, ProgramCycle
TITLE = "Main Program Sweep (Cycle)"
{ S7_Optimized_Access := 'TRUE' }
VERSION : 0.1
   VAR_INPUT
      Initial_Call : Bool;   // Initial call of this OB
      Remanence : Bool;   // =True, if remanent data are available
   END_VAR
BEGIN

REGION Network 1: Системный блок
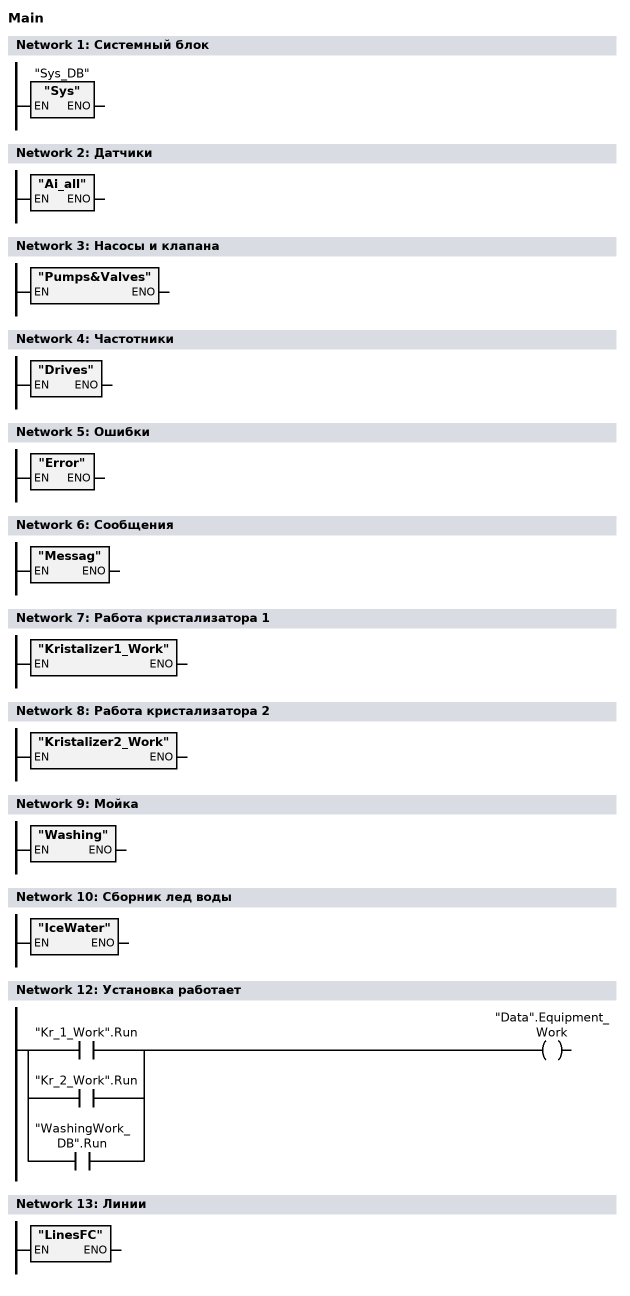
   RUNG wire#powerrail
      "Sys_DB"()
   END_RUNG
   // the same network as SCL:
   "Sys_DB"();   // "Sys"
END_REGION

REGION Network 2: Датчики
   RUNG wire#powerrail
      "Ai_all"()
   END_RUNG
   // the same network as SCL:
   "Ai_all"();
END_REGION

REGION Network 3: Насосы и клапана
   RUNG wire#powerrail
      "Pumps&Valves"()
   END_RUNG
   // the same network as SCL:
   "Pumps&Valves"();
END_REGION

REGION Network 4: Частотники
   RUNG wire#powerrail
      "Drives"()
   END_RUNG
   // the same network as SCL:
   "Drives"();
END_REGION

REGION Network 5: Ошибки
   RUNG wire#powerrail
      "Error"()
   END_RUNG
   // the same network as SCL:
   "Error"();
END_REGION

REGION Network 6: Сообщения
   RUNG wire#powerrail
      "Messag"()
   END_RUNG
   // the same network as SCL:
   "Messag"();
END_REGION

REGION Network 7: Работа кристализатора 1
   RUNG wire#powerrail
      "Kristalizer1_Work"()
   END_RUNG
   // the same network as SCL:
   "Kristalizer1_Work"();
END_REGION

REGION Network 8: Работа кристализатора 2
   RUNG wire#powerrail
      "Kristalizer2_Work"()
   END_RUNG
   // the same network as SCL:
   "Kristalizer2_Work"();
END_REGION

REGION Network 9: Мойка
   RUNG wire#powerrail
      "Washing"()
   END_RUNG
   // the same network as SCL:
   "Washing"();
END_REGION

REGION Network 10: Сборник лед воды
   RUNG wire#powerrail
      "IceWater"()
   END_RUNG
   // the same network as SCL:
   "IceWater"();
END_REGION

REGION Network 11 (SCL): Установка не работает и не в ручном закрыть все заслонки
   IF (NOT "Data".MAN_ON AND "Kr_1_Work"."Step" <> 1 AND "Kr_2_Work"."Step" <> 1 AND NOT "WashingWork_DB".Run)
       OR (("Kr_1_Work".Run OR "Kr_2_Work".Run OR "WashingWork_DB".Run)AND "Data".GlobalErrorStop) THEN
       "REG_Zero"();
   END_IF;
END_REGION

REGION Network 12: Установка работает
   RUNG wire#powerrail
      Contact( "Kr_1_Work".Run )
      wire#w1
      Coil( "Data".Equipment_Work )
   END_RUNG
   RUNG wire#powerrail
      Contact( "Kr_2_Work".Run )
   END_RUNG wire#w1
   RUNG wire#powerrail
      Contact( "WashingWork_DB".Run )
   END_RUNG wire#w1
   // the same network as SCL:
   "Data".Equipment_Work := "Kr_1_Work".Run OR "Kr_2_Work".Run OR "WashingWork_DB".Run;
END_REGION

REGION Network 13: Линии
   RUNG wire#powerrail
      "LinesFC"()
   END_RUNG
   // the same network as SCL:
   "LinesFC"();
END_REGION
END_ORGANIZATION_BLOCK

ORGANIZATION_BLOCK "Cyclic interrupt"   // OB30, LAD, CyclicInterrupt
{ S7_Optimized_Access := 'TRUE' }
VERSION : 0.1
   VAR_INPUT
      Initial_Call : Bool;   // Initial call of this OB
      Event_Count : Int;   // Events discarded
   END_VAR
BEGIN

REGION Network 1
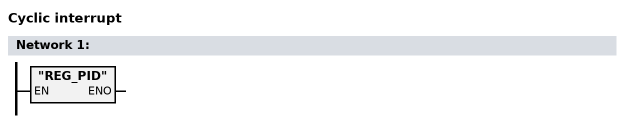
   RUNG wire#powerrail
      "REG_PID"()
   END_RUNG
   // the same network as SCL:
   "REG_PID"();
END_REGION
END_ORGANIZATION_BLOCK

ORGANIZATION_BLOCK "Time error interrupt"   // OB80, LAD, TimeErrorInterrupt
{ S7_Optimized_Access := 'TRUE' }
VERSION : 0.1
   VAR_INPUT
      Fault_ID : Byte;   // Fault identifier
      Csg_OBnr : OB_Any;   // Number of OB causing the error
      Csg_Prio : UInt;   // Priority of OB causing the error
   END_VAR
BEGIN
END_ORGANIZATION_BLOCK

ORGANIZATION_BLOCK "Diagnostic error interrupt"   // OB82, LAD, DiagnosticErrorInterrupt
{ S7_Optimized_Access := 'TRUE' }
VERSION : 0.1
   VAR_INPUT
      IO_State : Word;   // IO state of the HW object
      LADDR : Hw_Any;   // Hardware identifier
      Channel : UInt;   // Channel number
      MultiError : Bool;   // =true if more than one error is present
   END_VAR
BEGIN
END_ORGANIZATION_BLOCK

ORGANIZATION_BLOCK "Pull or plug of modules"   // OB83, LAD, PullPlug
{ S7_Optimized_Access := 'TRUE' }
VERSION : 0.1
   VAR_INPUT
      LADDR : Hw_Io;   // Hardware identifier
      Event_Class : Byte;   // 16#38/39: module inserted, removed
      Fault_ID : Byte;   // Fault identifier
   END_VAR
BEGIN
END_ORGANIZATION_BLOCK

ORGANIZATION_BLOCK "Rack or station failure"   // OB86, LAD, RackStationFailure
{ S7_Optimized_Access := 'TRUE' }
VERSION : 0.1
   VAR_INPUT
      LADDR : Hw_Device;   // Hardware identifier
      Event_Class : Byte;   // Event class
      Fault_ID : Byte;   // Fault identifier
   END_VAR
BEGIN
END_ORGANIZATION_BLOCK

ORGANIZATION_BLOCK "Programming error"   // OB121, LAD, ProgrammingError
{ S7_Optimized_Access := 'TRUE' }
VERSION : 0.1
   VAR_INPUT
      BlockNr : UInt;   // Number of causing block
      Reaction : USInt;   // 0:ignore, 1:substitute, 2:skip
      Fault_ID : Byte;   // Fault identifier
      BlockType : USInt;   // 16#01:OB, 16#02:FC, 16#03:FB, 16#04:SFC, 16#05:SFB, 16#06:DB: Type of block causing the error
      Area : USInt;   // Area where the error occured
      DBNr : DB_ANY;   // DB number if Area = DB or DI
      Csg_OBNr : OB_Any;   // Number of OB causing the error
      Csg_Prio : USInt;   // Priority of OB causing the error
      Width : USInt;   // 0:bit, 1:byte, 2:word, 3:dword, 4:lword
   END_VAR
BEGIN
END_ORGANIZATION_BLOCK

ORGANIZATION_BLOCK "IO access error"   // OB122, LAD, IOAccessError
{ S7_Optimized_Access := 'TRUE' }
VERSION : 0.1
   VAR_INPUT
      BlockNr : UInt;   // Number of causing block
      Reaction : USInt;   // 0:ignore, 1:substitute, 2:skip
      Fault_ID : Byte;   // 16#42:reading, 16#43:writing
      BlockType : USInt;   // 16#01:OB, 16#02:FC, 16#03:FB, 16#04:SFC, 16#05:SFB, 16#06:DB: Type of block causing the error
      Area : USInt;   // 16#81:I, 16#82:Q: IO area where the IOaccess error occured
      DBNr : DB_ANY;   // Reserved for system
      Csg_OBNr : OB_Any;   // Number of OB causing the error
      Csg_Prio : USInt;   // Priority of OB causing the error
      Width : USInt;   // 0:bit, 1:byte, 2:word, 3:dword, 4:lword
   END_VAR
BEGIN
END_ORGANIZATION_BLOCK

// folder: Ai

FUNCTION_BLOCK "ForVO"   // FB16, SCL
{ S7_Optimized_Access := 'FALSE' }
VERSION : 0.1
   VAR_INPUT
      Yi : Real;   // Текущее значение аналогового входного канала
      Ymax : Real := 0.0;   // Значение PIW/PID(Ai/Ad) при 100% входного диапазона
      Ymin : Real;   // Значение PIW/PID(Ai/Ad) при 0% входного диапазона
      Xmax : Real;   // Номинал Px при Ai=100%
      Xmin : Real;   // Номинал Px при Ai=0%
      Ke : Bool;   // Прямое использование канала
      Kf : Real;   // Коэффициент преобразования Ai=>Px (множитель)
      lag_koef : Real := 1.0;   // Множитель для сглаживания колебаний входного сигнала
      PV_AH_Lim : Real;   // Максимальний уровень сигнала
      PV_AL_Lim : Real;   // Минимальный уровень сигнала
      PV_WH_Lim : Real;   // Высокий уровень сигнала
      PV_WL_Lim : Real;   // Низкий уровень сигнала
      EnableAL_Lim : Bool := 1;
   END_VAR
   VAR_OUTPUT
      NDB : UDInt := 0;   // Номер InstanceDB
      Pz : Real;   // Фактическое значение канала
      Px : Real;   // Рабочее значение канала
      AH_LIM : Bool;
      AL_LIM : Bool;
   END_VAR
   VAR
      Alarm_error : Program_Alarm;
      Alarm_AH_Lim : Program_Alarm;
      Alarm_AL_Lim : Program_Alarm;
      Alarm_WH_Lim : Program_Alarm;
      Alarm_WL_Lim : Program_Alarm;
      ME : "DrvME";   // Набор данных для обработки ALARM_D
      initBlock : Bool;
      err : Bool;
   END_VAR
   VAR_TEMP
      Pu : Real;
      TSA : "TANY";   // Структура ANY для определения InstanceDB
      TPA AT TSA : ANY;   // Указатель ANY для определения InstanceDB
   END_VAR
BEGIN
   #err := (#Yi <= -32767 OR #Yi >= 32767);

   IF #Ymax - #Ymin <> 0 AND NOT #err THEN
       IF #Ke THEN
           #Pz := #Yi * #Kf+#Xmin;
       ELSE
           #Pz := (#Yi - #Ymin) / (#Ymax - #Ymin) * (#Xmax - #Xmin) + #Xmin;
       END_IF;
      // Сглаживание сигнала
       #Pu := #Pz;
       #Pu := (#Pu - #Px) * #lag_koef + #Px;
       #Px := #Pu;

       IF #Pz < #Xmin THEN
           #Pz := #Xmin;
       END_IF;

       IF #Px < #Xmin THEN
           #Px := #Xmin;
       END_IF;

   ELSE
       IF #Yi <= -32767 THEN
           #Pz := -99.0;
           #Px := -99.0;
       END_IF;

       IF #Yi >= 32767 THEN
           #Pz := 999.0;
           #Px := 999.0;
       END_IF;

       IF #Ymax - #Ymin = 0 THEN
           #Pz := -1.0;
           #Px := -1.0;
       END_IF;
   END_IF;


   // Запрос на инициализацию данных
   IF NOT #initBlock THEN
   // Инициализация данных
       #ME.Pr.N2 := 0;
       #ME.Pr.N3 := 0;
       #ME.Pr.N4 := 0;
       #ME.Pr.N5 := 0;
       #ME.Pr.N6 := 0;
   // Устанавливаем номер данного Instance Data Block
       #TPA := #ME;
       #NDB := #TSA.PTR.DN;
       #initBlock := 1;
   END_IF;


   // Сообщение: Неисправность канала датчика
   #ME.Pr.N1 := #NDB*10;
   #ME.Pr.N4 := #NDB*10;
   #Alarm_error(SIG := #err,
                TIMESTAMP := "TS0",
                SD_1:=#ME.Pr.N1, SD_2 := #ME.Pr.N4);


   // Сообщение: Максимальний уровень
   #AH_LIM := #Px > #PV_AH_Lim AND NOT #err;
   #Alarm_AH_Lim(SIG := #AH_LIM,
                  TIMESTAMP := "TS0",
                  SD_1 := #ME.Pr.N1, SD_2 := #ME.Pr.N4);

    // // Сообщение: Минимальный уровень
    #AL_LIM := #Px < #PV_AL_Lim AND NOT #err;
    #Alarm_AL_Lim(SIG :=#AL_LIM AND #EnableAL_Lim,
                  TIMESTAMP := "TS0",
                  SD_1 := #ME.Pr.N1, SD_2 := #ME.Pr.N4);

    // Сообщение: Высокий уровень
    // #Alarm_WH_Lim(SIG := #Px > #PV_WH_Lim AND NOT #err,
    //               TIMESTAMP := "TS0",
    //               SD_1 := #ME.Pr.N1);

    // Сообщение: Низкий уровень
    // #Alarm_WL_Lim(SIG := #Px < #PV_WL_Lim AND NOT #err,
    //               TIMESTAMP := "TS0",
    //               SD_1 := #ME.Pr.N1);
END_FUNCTION_BLOCK

FUNCTION "Ai_all" : Void   // FC2, SCL
{ S7_Optimized_Access := 'TRUE' }
VERSION : 0.1
   VAR_TEMP
      DelaTemp : Real;
   END_VAR
BEGIN
   // Температура TE1.1
   "AiCh_TE1.1"(Yi:="Ai_TE1.1",
                Xmax:=250.0,
                Xmin:=0,
                Ke:=1,
                Kf:=0.1,
                PV_AH_Lim:=105.0,
                EnableAL_Lim:=0);

   // Температура TE1.2
   "AiCh_TE1.2"(Yi:="Ai_TE1.2",
                Xmax:=250.0,
                Xmin:=0.0,
                Ke:=1,
                Kf:=0.1,
                PV_AH_Lim:=105.0);

   // Температура TE1.3
   "AiCh_TE1.3"(Yi:="Ai_TE1.3",
                Xmax:=250.0,
                Xmin:=0.0,
                Ke:=1,
                Kf:=0.1,
                PV_AH_Lim:=105.0,
                EnableAL_Lim:=0);

   // Температура TE2.1
   "AiCh_TE2.1"(Yi:="Ai_TE2.1",
                Xmax:=250.0,
                Xmin:=0.0,
                Ke:=1,
                Kf:=0.1,
                PV_AH_Lim:=105.0,
                EnableAL_Lim:=0);

   // Температура TE2.2
   "AiCh_TE2.2"(Yi:="Ai_TE2.2",
                Xmax:=250.0,
                Xmin:=0.0,
                Ke:=1,
                Kf:=0.1,
                PV_AH_Lim:=105.0,
                EnableAL_Lim:=0);

   // Температура TE2.3
   "AiCh_TE2.3"(Yi:="Ai_TE2.3",
                Xmax:=250.0,
                Xmin:=0.0,
                Ke:=1,
                Kf:=0.1,
                PV_AH_Lim:=105.0,
                EnableAL_Lim:=0);

   // Температура TE7.1
   "AiCh_TE7.1"(Yi:="Ai_TE7.1",
                Xmax:=250.0,
                Xmin:=0.0,
                Ke:=1,
                Kf:=0.1,
                PV_AH_Lim:=105.0,
                EnableAL_Lim:=0);

   // Температура TE7.2
   "AiCh_TE7.2"(Yi:="Ai_TE7.2",
                Xmax:=250.0,
                Xmin:=0.0,
                Ke:=1,
                Kf:=0.1,
                PV_AH_Lim:=105.0,
                EnableAL_Lim:=0);

   // Температура TE3.1
   // "AiCh_TE3.1"(Yi:="Ai_TE3.1",
   //              Xmax:=250.0,
   //              Xmin:=0.0,
   //              Ke:=1,
   //              Kf:=0.1,
   //              PV_AH_Lim:=105.0,
   //              PV_AL_Lim:=0.0);

   // // Температура TE3.2
   // "AiCh_TE3.2"(Yi:="Ai_TE3.2",
   //              Xmax:=250.0,
   //              Xmin:=0.0,
   //              Ke:=1,
   //              Kf:=0.1,
   //              PV_AH_Lim:=105.0,
   //              EnableAL_Lim:=0);

   // // Температура TE3.3
   // "AiCh_TE3.3"(Yi:="Ai_TE3.3",
   //              Xmax:=250.0,
   //              Xmin:=0.0,
   //              Ke:=1,
   //              Kf:=0.1,
   //              PV_AH_Lim:=105.0,
   //              EnableAL_Lim:=0);

   //------------------------------------------ Уровни--------------------

   // Уровень LIC 1.1
   "AiCh_LIC1.1"(Yi:="Ai_LIC1.1",
                 Xmax:=100.0,
                 Xmin:=0.0,
                 PV_AH_Lim:=105.0,
                 EnableAL_Lim:=0);

   // Уровень LIC 2.1
    "AiCh_LIC2.1"(Yi:="Ai_LIC2.1",
                  Xmax:=100.0,
                  Xmin:=0.0,
                  PV_AH_Lim:=105.0,
                  EnableAL_Lim:=0);

    // Уровень LIC 3.1
    // "AiCh_LIC3.1"(Yi:="Ai_LIC3.1",
    //               Xmax:=100.0,
    //               Xmin:=0.0,
    //               PV_AH_Lim:=105.0,
    //               EnableAL_Lim:=0);

    // Уровень LIC 7.1
    "AiCh_LIC7.1"(Yi := "Ai_LIC7.1",
                  Xmax := 1.0,
                  Xmin := -1.0,
                  PV_AH_Lim := 105.0,
                  EnableAL_Lim:=0);

    // Уровень LIC 7.2
    "AiCh_LIC7.2"(Yi:="Ai_LIC7.2",
                  Xmax:=1.0,
                  Xmin:=-1.0,
                  PV_AH_Lim:=105.0,
                  EnableAL_Lim:=0);


    //---------------------- Уровень в ВО-------------------------------------
     #DelaTemp := "AiCh_LIC7.2".Px - "AiCh_LIC7.1".Px;

    "ForVO_DB"(Yi:= #DelaTemp,
               Ymax:=1.0,
               Ymin:=-1.0,
               Xmax:=100.0,
               PV_AH_Lim:=105.0,
               EnableAL_Lim:=0);



    "Data".LevelVO_Pv :=  "ForVO_DB".Px;
END_FUNCTION

// folder: Drives

FUNCTION "Drives" : Void   // FC3, LAD
{ S7_Optimized_Access := 'TRUE' }
VERSION : 0.1
   VAR_TEMP
      M1_1_Vs : Real;
      M2_1_Vs : Real;
   END_VAR
BEGIN

REGION Network 1 (SCL): Ручной режим
   IF "Data".MAN_ON THEN
       #M1_1_Vs := "Data".Mixer1.Man;
       #M2_1_Vs := "Data".Mixer2.Man;
   ELSE
       #M1_1_Vs := "Mixer1_Work_DB".PowerOut;
       #M2_1_Vs := "Mixer2_Work_DB".PowerOut;
   END_IF;
END_REGION

REGION Network 2: Частотник M1_1
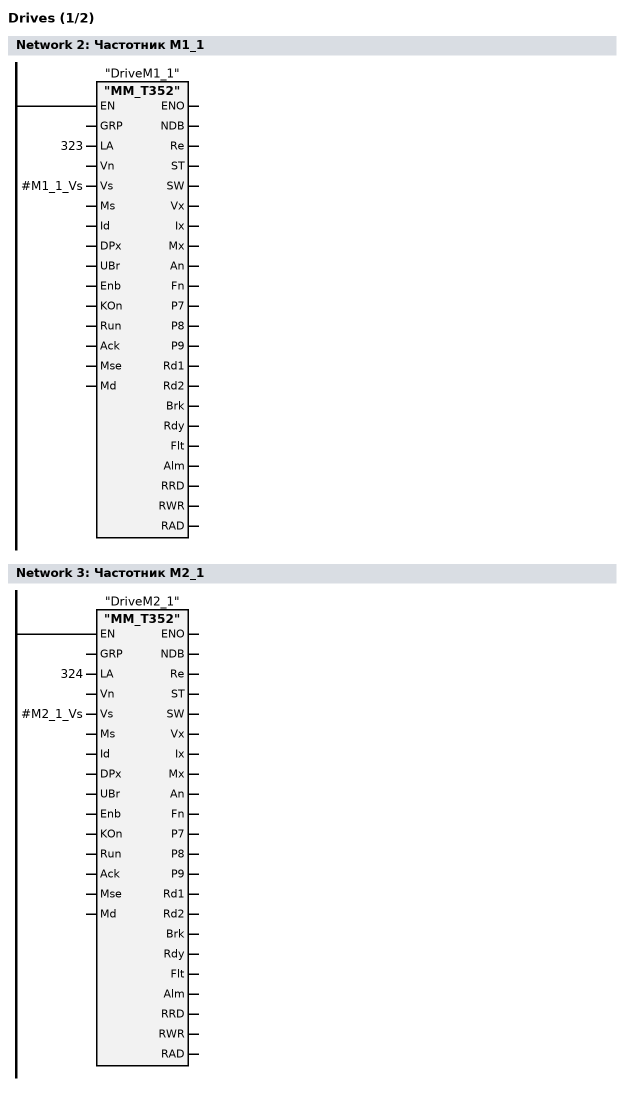
   RUNG wire#powerrail
      "DriveM1_1"(GRP :=, LA := 323, Vn :=, Vs := #M1_1_Vs, Ms :=, Id :=, DPx :=, UBr :=, Enb :=, KOn :=, Run :=, Ack :=, Mse :=, Md :=, NDB =>, Re =>, ST =>, SW =>, Vx =>, Ix =>, Mx =>, An =>, Fn =>, P7 =>, P8 =>, P9 =>, Rd1 =>, Rd2 =>, Brk =>, Rdy =>, Flt =>, Alm =>, RRD =>, RWR =>, RAD =>)
   END_RUNG
   // the same network as SCL:
   "DriveM1_1"(LA := 323, Vs := #M1_1_Vs);   // "MM_T352"
END_REGION

REGION Network 3: Частотник M2_1
   RUNG wire#powerrail
      "DriveM2_1"(GRP :=, LA := 324, Vn :=, Vs := #M2_1_Vs, Ms :=, Id :=, DPx :=, UBr :=, Enb :=, KOn :=, Run :=, Ack :=, Mse :=, Md :=, NDB =>, Re =>, ST =>, SW =>, Vx =>, Ix =>, Mx =>, An =>, Fn =>, P7 =>, P8 =>, P9 =>, Rd1 =>, Rd2 =>, Brk =>, Rdy =>, Flt =>, Alm =>, RRD =>, RWR =>, RAD =>)
   END_RUNG
   // the same network as SCL:
   "DriveM2_1"(LA := 324, Vs := #M2_1_Vs);   // "MM_T352"
END_REGION

REGION Network 4: Частотник M7_1
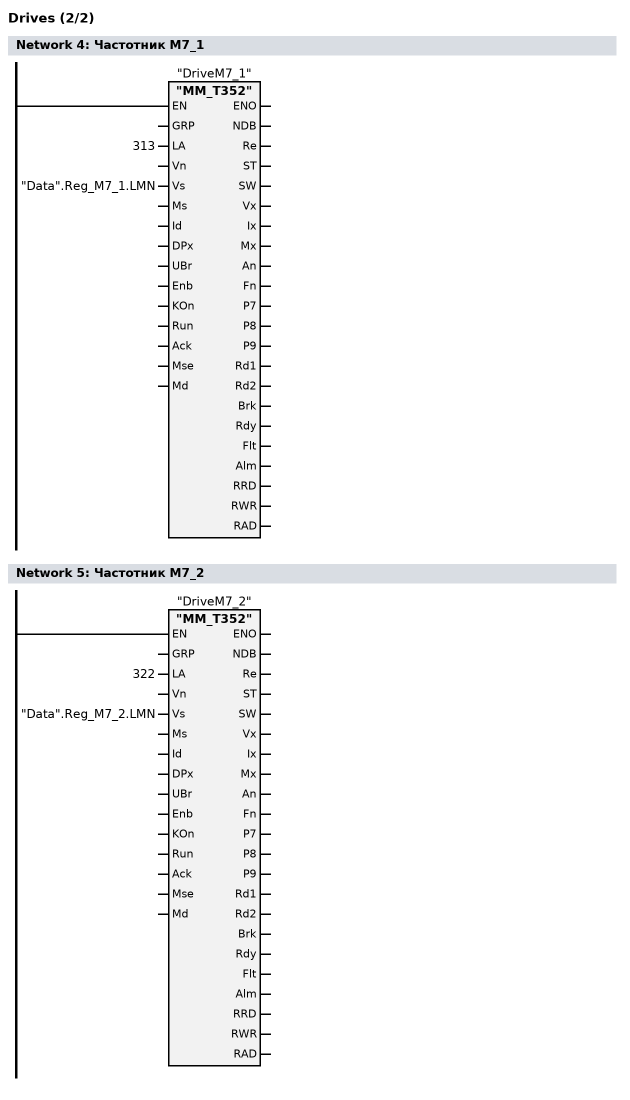
   RUNG wire#powerrail
      "DriveM7_1"(GRP :=, LA := 313, Vn :=, Vs := "Data".Reg_M7_1.LMN, Ms :=, Id :=, DPx :=, UBr :=, Enb :=, KOn :=, Run :=, Ack :=, Mse :=, Md :=, NDB =>, Re =>, ST =>, SW =>, Vx =>, Ix =>, Mx =>, An =>, Fn =>, P7 =>, P8 =>, P9 =>, Rd1 =>, Rd2 =>, Brk =>, Rdy =>, Flt =>, Alm =>, RRD =>, RWR =>, RAD =>)
   END_RUNG
   // the same network as SCL:
   "DriveM7_1"(LA := 313, Vs := "Data".Reg_M7_1.LMN);   // "MM_T352"
END_REGION

REGION Network 5: Частотник M7_2
   RUNG wire#powerrail
      "DriveM7_2"(GRP :=, LA := 322, Vn :=, Vs := "Data".Reg_M7_2.LMN, Ms :=, Id :=, DPx :=, UBr :=, Enb :=, KOn :=, Run :=, Ack :=, Mse :=, Md :=, NDB =>, Re =>, ST =>, SW =>, Vx =>, Ix =>, Mx =>, An =>, Fn =>, P7 =>, P8 =>, P9 =>, Rd1 =>, Rd2 =>, Brk =>, Rdy =>, Flt =>, Alm =>, RRD =>, RWR =>, RAD =>)
   END_RUNG
   // the same network as SCL:
   "DriveM7_2"(LA := 322, Vs := "Data".Reg_M7_2.LMN);   // "MM_T352"
END_REGION
END_FUNCTION

// folder: Errors

FUNCTION "Error" : Void   // FC4, LAD
{ S7_Optimized_Access := 'TRUE' }
VERSION : 0.1
BEGIN

REGION Network 1 (SCL): Ошибки
   // Ошибки аналоговых датчиков
   "FpDW_DB".F[0] := "AiCh_TE1.1".err;
   "FpDW_DB".F[1] := "AiCh_TE1.2".err;
   "FpDW_DB".F[2] := "AiCh_TE1.3".err;
   "FpDW_DB".F[3] := "AiCh_TE2.1".err;
   "FpDW_DB".F[4] := "AiCh_TE2.2".err;
   "FpDW_DB".F[5] := "AiCh_TE2.3".err;
   "FpDW_DB".F[6] := "AiCh_TE7.1".err;
   "FpDW_DB".F[7] := "AiCh_TE7.2".err;
   "FpDW_DB".F[8] := "AiCh_TE3.1".err;
   "FpDW_DB".F[9] := "AiCh_TE3.2".err;
   "FpDW_DB".F[10] := "AiCh_LIC1.1".err;
   "FpDW_DB".F[11] := "AiCh_LIC2.1".err;
   "FpDW_DB".F[12] := "AiCh_LIC3.1".err;
   "FpDW_DB".F[13] := "AiCh_LIC7.1".err;
   "FpDW_DB".F[14] := "AiCh_LIC7.2".err;

   // Ошибки насосов и клапанов
   "FpDW_DB".F[15] := "DrvCell_M1_1".Err;
   "FpDW_DB".F[16] := "DrvCell_M1_2".Err;
   "FpDW_DB".F[17] := "DrvCell_M2_1".Err;
   "FpDW_DB".F[18] := "DrvCell_M2_2".Err;
   "FpDW_DB".F[19] := "DrvCell_M3".Err;
   "FpDW_DB".F[20] := "DrvCell_M4".Err;
   "FpDW_DB".F[21] := "DrvCell_M7_1".Err;
   "FpDW_DB".F[22] := "DrvCell_M7_2".Err;
   "FpDW_DB".F[23] := "DrvCell_M10".Err;
   "FpDW_DB".F[24] := "DrvCell_V7_1".Err;
   "FpDW_DB".F[25] := "DrvCell_V7_2".Err;
   "FpDW_DB".F[26] := "DrvCell_V1_1".Err;
   "FpDW_DB".F[27] := "DrvCell_V2_1".Err;
   "FpDW_DB".F[28] := "DrvCell_V3_1".Err;
   "FpDW_DB".F[29] := "DrvCell_V1_7".Err;
   "FpDW_DB".F[30] := "DrvCell_V2_7".Err;
   "FpDW_DB".F[31] := "DrvCell_V3_7".Err;
   "FpDW_DB".F[32] := "DrvCell_V7_3".Err;
   "FpDW_DB".F[33] := "DrvCell_V7_4".Err;



   // Ошибки другие
   "FpDW_DB".F[34] := NOT "Di_AvarStop";
   "FpDW_DB".F[35] := NOT "Di_KF01";
   "FpDW_DB".F[36] := NOT "Di_Ksp01";
   "FpDW_DB".F[37] := NOT  "Di_Lah1.1";
   "FpDW_DB".F[38] := NOT  "Di_Lah2.1";
   "FpDW_DB".F[39] := 0;
   "FpDW_DB".F[40] := NOT "Di_Ga1.4"  AND ("Kr_1_Work".Run OR "WashingWork_DB"."Step"=3);
   "FpDW_DB".F[41] :=  NOT "Di_Ga2.4" AND ("Kr_2_Work".Run OR "WashingWork_DB"."Step"=4);


   "FpDW_DB"();

   "Data".Erorrs_Beep := "FpDW_DB".Fe;
END_REGION

REGION Network 2: Глобальная ошибка
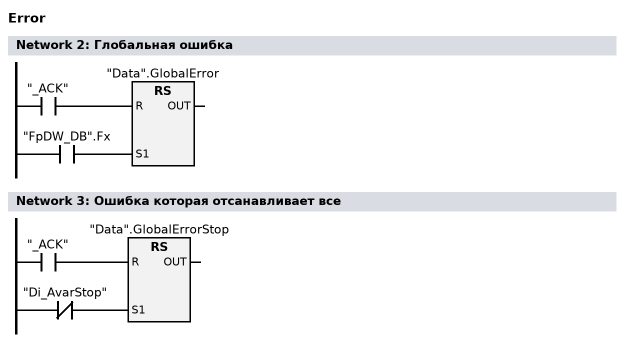
   RUNG wire#powerrail
      Contact( "_ACK" )
      S_RS(operand := "Data".GlobalError, s1 := wire#w1)
   END_RUNG
   RUNG wire#powerrail
      Contact( "FpDW_DB".Fx )
   END_RUNG wire#w1
   // the same network as SCL:
   IF "_ACK" THEN
       "Data".GlobalError := FALSE;   // RS flip-flop
   END_IF;
   IF "FpDW_DB".Fx THEN "Data".GlobalError := TRUE; END_IF;
END_REGION

REGION Network 3: Ошибка которая отсанавливает все
   RUNG wire#powerrail
      Contact( "_ACK" )
      S_RS(operand := "Data".GlobalErrorStop, s1 := wire#w1)
   END_RUNG
   RUNG wire#powerrail
      I_Contact( "Di_AvarStop" )
   END_RUNG wire#w1
   // the same network as SCL:
   IF "_ACK" THEN
       "Data".GlobalErrorStop := FALSE;   // RS flip-flop
   END_IF;
   IF NOT "Di_AvarStop" THEN "Data".GlobalErrorStop := TRUE; END_IF;
END_REGION
END_FUNCTION

// folder: Flip

FUNCTION_BLOCK "FlipSingle"   // FB5, LAD
{ S7_Optimized_Access := 'TRUE' }
VERSION : 0.1
   VAR_INPUT
      in : Bool;
      Time_pause : DInt;
      Time_work : DInt;
   END_VAR
   VAR_OUTPUT
      out : Bool;
   END_VAR
   VAR
      TimeWorkMs : Time;
      TimeResetMs : Time;
      Timer_pause : TON_TIME;
      Timer_work : TP_TIME;
      Timer_Num : Int;
      Front : R_TRIG;
      NegFront : F_TRIG;
   END_VAR
BEGIN

REGION Network 1 (SCL)
   #Front(CLK := #in);
   #NegFront(CLK := #in);

   IF #Front.Q THEN
       #Timer_Num := 1;
   END_IF;

   IF #NegFront.Q THEN
       #Timer_Num := 0;
   END_IF;



   CASE #Timer_Num OF
       1:
           #Timer_pause(IN:=TRUE,PT:=T_CONV(#Time_pause*1000),Q=>#out);
           #Timer_work(IN :=  #Timer_pause.Q,
                         PT := T_CONV(#Time_work*1000));
             IF NOT #Timer_work.Q AND #Timer_pause.Q THEN
               #out := false;
               RESET_TIMER(#Timer_pause);
           END_IF;
       ELSE
           #out := false;
           RESET_TIMER(#Timer_pause);

   END_CASE;
END_REGION
END_FUNCTION_BLOCK

// folder: IceWater

FUNCTION_BLOCK "IceWaterWork"   // FB8, SCL
{ S7_Optimized_Access := 'TRUE' }
VERSION : 0.1
   VAR_INPUT
      AvarStop : Bool;
      Top : Bool;
      Bottom : Bool;
   END_VAR
   VAR_OUTPUT
      M3 : Bool;
   END_VAR
BEGIN


   IF NOT #AvarStop THEN
       IF #Top THEN
           #M3 := TRUE;

           // Нижний уровень сборника
       ELSIF NOT #Bottom THEN
           #M3 := FALSE;
       END_IF;

   ELSE
       #M3 := FALSE;
   END_IF;
END_FUNCTION_BLOCK

FUNCTION "IceWater" : Void   // FC9, LAD
{ S7_Optimized_Access := 'TRUE' }
VERSION : 0.1
BEGIN

REGION Network 1: Работа сборника лед - воды
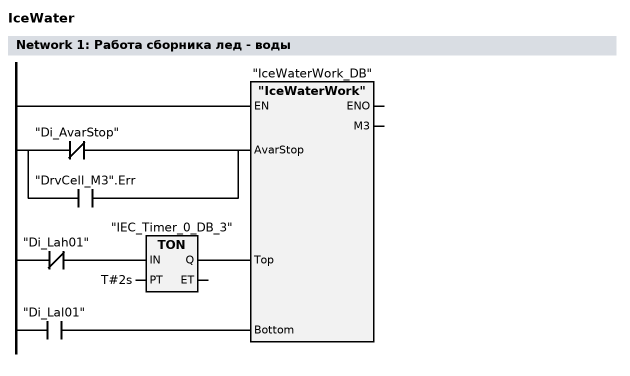
   "IEC_Timer_0_DB_3".TON(IN := NOT "Di_Lah01", PT := T#2s);
   "IceWaterWork_DB"(AvarStop := NOT "Di_AvarStop" OR "DrvCell_M3".Err,   // "IceWaterWork"
                     Top := "IEC_Timer_0_DB_3".Q,
                     Bottom := "Di_Lal01");
END_REGION
END_FUNCTION

// folder: KristalizersWork

FUNCTION_BLOCK "MixerWork"   // FB2, SCL
{ S7_Optimized_Access := 'TRUE' }
VERSION : 0.1
   VAR_INPUT
      Start : Bool;
      PowerIn : Real;
      RegimBothSide : Bool;
      TimeRight : DInt;
      TimeLeft : DInt;
      TimePause : DInt;
      AvariyStop : Bool;
   END_VAR
   VAR_OUTPUT
      Motor : Bool;
      PowerOut : Real;
   END_VAR
   VAR
      Run : Bool;
      TimerRight : TONR_TIME;
      TimerLeft : TONR_TIME;
      TimerPause : TONR_TIME;
      TimerNum : Int;
      TimerNumPrev : Int;
      FrontStart : R_TRIG;
   END_VAR
BEGIN
   // Включаем миксер

   #FrontStart(CLK := #Start);

   IF #FrontStart.Q THEN
       #Run := TRUE;
       #TimerNum := 1;
   END_IF;


   IF NOT #Start THEN 
       #Run := FALSE;
   END_IF;



   IF #Run AND NOT #AvariyStop THEN

       IF #RegimBothSide THEN
           CASE #TimerNum OF
               1: // Режим Вправо
                   #Motor := TRUE;
                   #PowerOut := #PowerIn;
                   #TimerNumPrev := 1;


                   #TimerRight(IN := TRUE,
                               PT := T_CONV(#TimeRight * 1000));

                   IF #TimerRight.Q THEN
                       #TimerNum := 2;
                       RESET_TIMER(#TimerRight);
                   END_IF;

               2: // Режим пауза
                   #Motor := FALSE;
                   #PowerOut := 0.0;

                   #TimerPause(IN:=TRUE, PT:=T_CONV(#TimePause*1000));

                   IF #TimerPause.Q THEN

                       IF #TimerNumPrev = 1 THEN
                           #TimerNum := 3;

                       ELSIF #TimerNumPrev = 3 THEN
                           #TimerNum := 1;

                       END_IF;

                       RESET_TIMER(#TimerPause);

                  END_IF;

              3: // Режим влево
                  #Motor := TRUE;
                  #PowerOut := #PowerIn * -1;
                  #TimerNumPrev := 3;

                  #TimerLeft(IN := TRUE,
                             PT := T_CONV(#TimeLeft * 1000));

                  IF #TimerLeft.Q THEN
                      #TimerNum := 2;
                      RESET_TIMER(#TimerLeft);
                  END_IF;

           END_CASE;

       ELSE
           #TimerNum := 1;
           RESET_TIMER(#TimerRight);
           RESET_TIMER(#TimerPause);
           RESET_TIMER(#TimerLeft);
           #Motor := TRUE;
           #PowerOut := #PowerIn;

       END_IF;

   ELSE
       #Motor := FALSE;
       #PowerOut := 0.0;
       #TimerRight.IN := FALSE;
       #TimerPause.IN := FALSE;
       #TimerLeft.IN := FALSE;

       IF NOT #AvariyStop OR NOT #Run THEN
           RESET_TIMER(#TimerRight);
           RESET_TIMER(#TimerPause);
           RESET_TIMER(#TimerLeft);
           #TimerNumPrev := 1;
       END_IF;
   END_IF;
END_FUNCTION_BLOCK

FUNCTION_BLOCK "KristalizerWork"   // FB13, SCL
{ S7_Optimized_Access := 'TRUE' }
VERSION : 0.1
   VAR_INPUT
      StepDesition : Int := 1;
      Start : Bool;
      Stop : Bool;
      TempInSp : Real;
      Power_M7_2 : Real;
      TempFillingSP : Real;
      TempKristSP : Real;
      TimeKristal_min : DInt;
      TempKristPV : Real;
      LevelTop : Real;
      LevelBotoom : Real;
      LevelPV : Real;
      AvariyStop : Bool;
   END_VAR
   VAR_OUTPUT
      Mixer : Bool;
      V7_3 : Bool;
      M7_1 : Bool;
      M7_2 : Bool;
      M10 : Bool;
      "M1_2/2_2" : Bool;
      M5 : Bool;
      Beep : Bool;
      TE_Kristal_in : Bool;
      TE_Kristal_SP : Real;
      LeftTimeMin : DInt;
   END_VAR
   VAR
      Run : Bool;
      FrontStart : R_TRIG;
      FrontStop : R_TRIG;
      "Step" : Int;
      LevelTop_Stat : Bool;
      TempSec : Real;
      TempHour : Real;
      "Timer" : TONR_TIME;
      TimerTop : TON_TIME;
      TimerBottom : TON_TIME;
      SecondPassed : DInt;
   END_VAR
BEGIN
   #FrontStart(CLK := #Start);
   #FrontStop(CLK := #Stop);

   IF #FrontStart.Q THEN
       #Run := TRUE;
       #"Step" := #StepDesition;
   END_IF;

   IF #FrontStop.Q THEN
       #Run := FALSE;
   END_IF;


   IF #Run AND NOT #AvariyStop THEN
       // Включаем миксер
       #Mixer:=TRUE;

       CASE #"Step" OF

           1: // Набор продукта

               #V7_3 := TRUE;

               // Заслонка 1RV01
               "Data".Reg_01RV01.Man_On := FALSE;


               // Насос продукта
               "Data".Reg_M7_1.Man_On := FALSE;

               #M7_1 := TRUE;

               // Насос M10
               #M10 := TRUE;

               // Насос вакуумный 
               "Data".Reg_M7_2.Man_On := TRUE;
               "Data".Reg_M7_2.Man := #Power_M7_2;
               #M7_2 := TRUE;

               #"M1_2/2_2" := TRUE;

               #TE_Kristal_SP := #TempFillingSP;
               #TE_Kristal_in := TRUE;

               #TimerTop(IN := #LevelPV >= #LevelTop,
                         PT := T#2s);

               IF #TimerTop.Q  AND NOT #LevelTop_Stat THEN
                   #Beep := TRUE;
                   #LevelTop_Stat := TRUE;
               END_IF;


           2: // Кристализация продукта
               // Высчитываем убывание температуры за секунду
               #TempSec := (#TempFillingSP - #TempKristSP) / (#TimeKristal_min * 60);
               #"Timer"(IN := TRUE,
                      PT := T_CONV(#TimeKristal_min * 60000));

               #SecondPassed := #"Timer".ET / 1000;

               #TE_Kristal_in:=TRUE;
               #TE_Kristal_SP := (#TempFillingSP - (#TempSec * #SecondPassed));

               #LeftTimeMin := (T_CONV(#TimeKristal_min * 60000) - #"Timer".ET) / 60000;

               #"M1_2/2_2" := TRUE;

           3: // Выдача продукта

               #M5 := TRUE;

               #TimerBottom(IN:=#LevelPV < #LevelBotoom, PT:=T#2s);


               IF  #TimerBottom.Q AND NOT #LevelTop_Stat THEN
                   #Beep := TRUE;
                   #LevelTop_Stat := TRUE;
               END_IF;



       END_CASE;

   ELSE

       #"Timer".IN := FALSE;
       IF NOT #AvariyStop OR NOT #Run THEN
           RESET_TIMER(#"Timer");
           #LevelTop_Stat := FALSE;
           #LeftTimeMin := 0;
           #"Step" := 0;
       END_IF;


       #Mixer := FALSE;
       #V7_3 := FALSE;
       #M7_1 := FALSE;
       #M7_2 := FALSE;

       RESET_TIMER(#TimerTop);
       RESET_TIMER(#TimerBottom);

       #M10 := FALSE;
       #"M1_2/2_2" := FALSE;

       #M5 := FALSE;

       #TE_Kristal_in := FALSE;

       #TempSec := 0;
       #SecondPassed := 0;



   END_IF;


   IF "_ACK" THEN
       #Beep := FALSE;
   END_IF;

   // Высчитываем скорость температуры в час
   #TempHour := (#TempFillingSP - #TempKristSP) / #TimeKristal_min;
END_FUNCTION_BLOCK

FUNCTION "Kristalizer1_Work" : Void   // FC10, LAD
{ S7_Optimized_Access := 'TRUE' }
VERSION : 0.1
   VAR_TEMP   // added for the SCL form of the ladder/FBD networks
      _w1 : Bool;
      _w2 : Bool;
      _w3 : Bool;
   END_VAR
BEGIN

REGION Network 1: Готовность маршрута
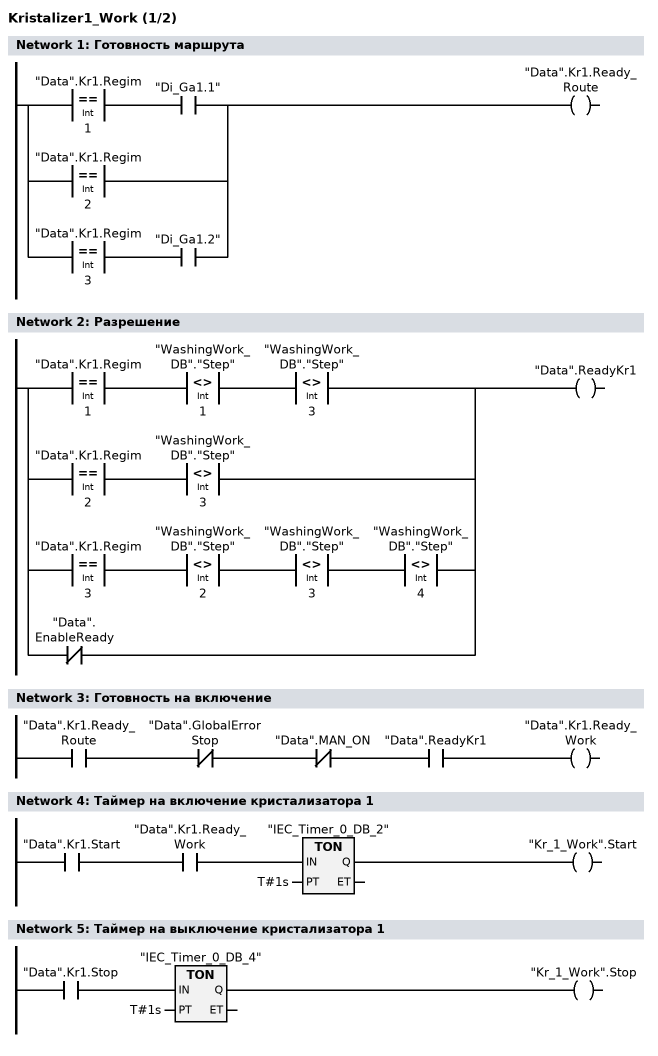
   RUNG wire#powerrail
      { S7_Templates := "SrcType := Int" } EQ_Contact(in1 := "Data".Kr1.Regim, in2 := 1)
      Contact( "Di_Ga1.1" )
      wire#w1
      Coil( "Data".Kr1.Ready_Route )
   END_RUNG
   RUNG wire#powerrail
      { S7_Templates := "SrcType := Int" } EQ_Contact(in1 := "Data".Kr1.Regim, in2 := 2)
   END_RUNG wire#w1
   RUNG wire#powerrail
      { S7_Templates := "SrcType := Int" } EQ_Contact(in1 := "Data".Kr1.Regim, in2 := 3)
      Contact( "Di_Ga1.2" )
   END_RUNG wire#w1
   // the same network as SCL:
   "Data".Kr1.Ready_Route := (("Data".Kr1.Regim = 1) AND "Di_Ga1.1") OR ("Data".Kr1.Regim = 2) OR (("Data".Kr1.Regim = 3) AND "Di_Ga1.2");
END_REGION

REGION Network 2: Разрешение
   RUNG wire#powerrail
      { S7_Templates := "SrcType := Int" } EQ_Contact(in1 := "Data".Kr1.Regim, in2 := 1)
      { S7_Templates := "SrcType := Int" } NE_Contact(in1 := "WashingWork_DB"."Step", in2 := 1)
      { S7_Templates := "SrcType := Int" } NE_Contact(in1 := "WashingWork_DB"."Step", in2 := 3)
      wire#w1
      Coil( "Data".ReadyKr1 )
   END_RUNG
   RUNG wire#powerrail
      { S7_Templates := "SrcType := Int" } EQ_Contact(in1 := "Data".Kr1.Regim, in2 := 2)
      { S7_Templates := "SrcType := Int" } NE_Contact(in1 := "WashingWork_DB"."Step", in2 := 3)
   END_RUNG wire#w1
   RUNG wire#powerrail
      { S7_Templates := "SrcType := Int" } EQ_Contact(in1 := "Data".Kr1.Regim, in2 := 3)
      { S7_Templates := "SrcType := Int" } NE_Contact(in1 := "WashingWork_DB"."Step", in2 := 2)
      { S7_Templates := "SrcType := Int" } NE_Contact(in1 := "WashingWork_DB"."Step", in2 := 3)
      { S7_Templates := "SrcType := Int" } NE_Contact(in1 := "WashingWork_DB"."Step", in2 := 4)
   END_RUNG wire#w1
   RUNG wire#powerrail
      I_Contact( "Data".EnableReady )
   END_RUNG wire#w1
   // the same network as SCL:
   "Data".ReadyKr1 := (("Data".Kr1.Regim = 1) AND ("WashingWork_DB"."Step" <> 1) AND ("WashingWork_DB"."Step" <> 3)) OR (("Data".Kr1.Regim = 2) AND ("WashingWork_DB"."Step" <> 3)) OR (("Data".Kr1.Regim = 3) AND ("WashingWork_DB"."Step" <> 2) AND ("WashingWork_DB"."Step" <> 3) AND ("WashingWork_DB"."Step" <> 4)) OR NOT "Data".EnableReady;
END_REGION

REGION Network 3: Готовность на включение
   RUNG wire#powerrail
      Contact( "Data".Kr1.Ready_Route )
      I_Contact( "Data".GlobalErrorStop )
      I_Contact( "Data".MAN_ON )
      Contact( "Data".ReadyKr1 )
      Coil( "Data".Kr1.Ready_Work )
   END_RUNG
   // the same network as SCL:
   "Data".Kr1.Ready_Work := "Data".Kr1.Ready_Route AND NOT "Data".GlobalErrorStop AND NOT "Data".MAN_ON AND "Data".ReadyKr1;
END_REGION

REGION Network 4: Таймер на включение кристализатора 1
   "IEC_Timer_0_DB_2".TON(IN := "Data".Kr1.Start AND "Data".Kr1.Ready_Work, PT := T#1s);
   "Kr_1_Work".Start := "IEC_Timer_0_DB_2".Q;
END_REGION

REGION Network 5: Таймер на выключение кристализатора 1
   "IEC_Timer_0_DB_4".TON(IN := "Data".Kr1.Stop, PT := T#1s);
   "Kr_1_Work".Stop := "IEC_Timer_0_DB_4".Q;
END_REGION

REGION Network 6: Работа кристализатора №1
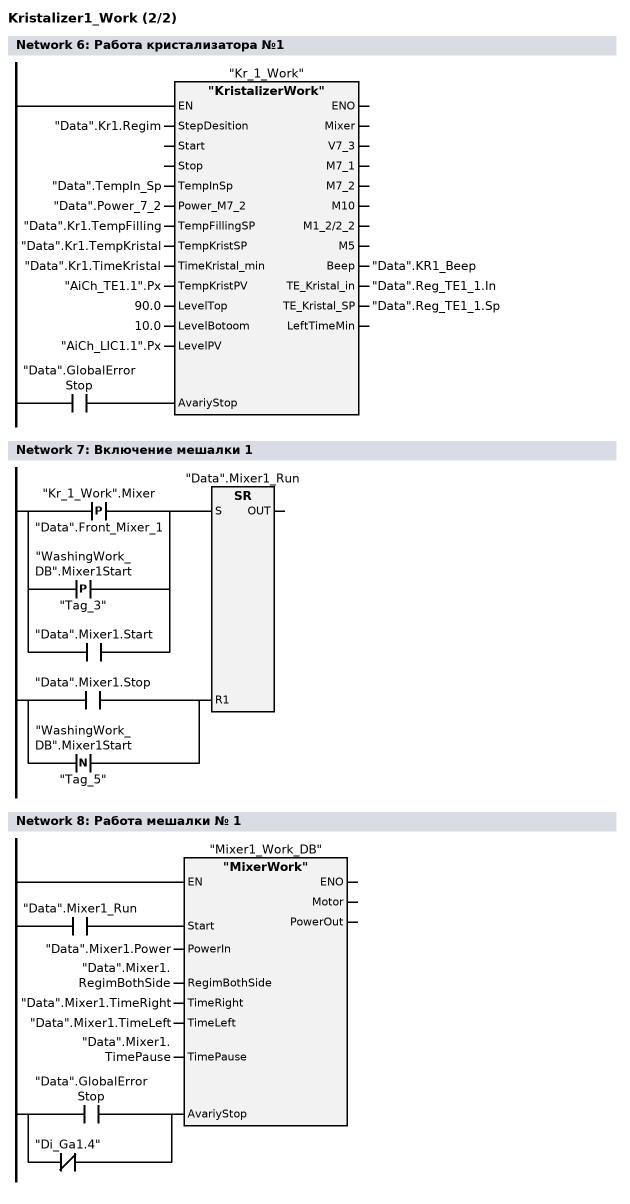
   RUNG wire#powerrail
      "Kr_1_Work"(AvariyStop := wire#w1, StepDesition := "Data".Kr1.Regim, Start :=, Stop :=, TempInSp := "Data".TempIn_Sp, Power_M7_2 := "Data".Power_7_2, TempFillingSP := "Data".Kr1.TempFilling, TempKristSP := "Data".Kr1.TempKristal, TimeKristal_min := "Data".Kr1.TimeKristal, TempKristPV := "AiCh_TE1.1".Px, LevelTop := 90.0, LevelBotoom := 10.0, LevelPV := "AiCh_LIC1.1".Px, Mixer =>, V7_3 =>, M7_1 =>, M7_2 =>, M10 =>, "M1_2/2_2" =>, M5 =>, Beep => "Data".KR1_Beep, TE_Kristal_in => "Data".Reg_TE1_1.In, TE_Kristal_SP => "Data".Reg_TE1_1.Sp, LeftTimeMin =>)
   END_RUNG
   RUNG wire#powerrail
      Contact( "Data".GlobalErrorStop )
   END_RUNG wire#w1
   // the same network as SCL:
   "Kr_1_Work"(StepDesition := "Data".Kr1.Regim,   // "KristalizerWork"
               TempInSp := "Data".TempIn_Sp,
               Power_M7_2 := "Data".Power_7_2,
               TempFillingSP := "Data".Kr1.TempFilling,
               TempKristSP := "Data".Kr1.TempKristal,
               TimeKristal_min := "Data".Kr1.TimeKristal,
               TempKristPV := "AiCh_TE1.1".Px,
               LevelTop := 90.0,
               LevelBotoom := 10.0,
               LevelPV := "AiCh_LIC1.1".Px,
               AvariyStop := "Data".GlobalErrorStop,
               Beep => "Data".KR1_Beep,
               TE_Kristal_in => "Data".Reg_TE1_1.In,
               TE_Kristal_SP => "Data".Reg_TE1_1.Sp);
END_REGION

REGION Network 7: Включение мешалки 1
   RUNG wire#powerrail
      P_Contact(operand := "Kr_1_Work".Mixer, bit := "Data".Front_Mixer_1)
      wire#w1
      S_SR(operand := "Data".Mixer1_Run, r1 := wire#w2)
   END_RUNG
   RUNG wire#powerrail
      P_Contact(operand := "WashingWork_DB".Mixer1Start, bit := "Tag_3")
   END_RUNG wire#w1
   RUNG wire#powerrail
      Contact( "Data".Mixer1.Start )
   END_RUNG wire#w1
   RUNG wire#powerrail
      Contact( "Data".Mixer1.Stop )
   END_RUNG wire#w2
   RUNG wire#powerrail
      N_Contact(operand := "WashingWork_DB".Mixer1Start, bit := "Tag_5")
   END_RUNG wire#w2
   // the same network as SCL:
   #_w1 := "Kr_1_Work".Mixer AND NOT "Data".Front_Mixer_1;   // rising edge of "Kr_1_Work".Mixer
   "Data".Front_Mixer_1 := "Kr_1_Work".Mixer;
   #_w2 := "WashingWork_DB".Mixer1Start AND NOT "Tag_3";   // rising edge of "WashingWork_DB".Mixer1Start
   "Tag_3" := "WashingWork_DB".Mixer1Start;
   #_w3 := NOT "WashingWork_DB".Mixer1Start AND "Tag_5";   // falling edge of "WashingWork_DB".Mixer1Start
   "Tag_5" := "WashingWork_DB".Mixer1Start;
   IF #_w1 OR #_w2 OR "Data".Mixer1.Start THEN
       "Data".Mixer1_Run := TRUE;   // SR flip-flop
   END_IF;
   IF "Data".Mixer1.Stop OR #_w3 THEN "Data".Mixer1_Run := FALSE; END_IF;
END_REGION

REGION Network 8: Работа мешалки № 1
   RUNG wire#powerrail
      "Mixer1_Work_DB"(Start := wire#w1, AvariyStop := wire#w2, PowerIn := "Data".Mixer1.Power, RegimBothSide := "Data".Mixer1.RegimBothSide, TimeRight := "Data".Mixer1.TimeRight, TimeLeft := "Data".Mixer1.TimeLeft, TimePause := "Data".Mixer1.TimePause, Motor =>, PowerOut =>)
   END_RUNG
   RUNG wire#powerrail
      Contact( "Data".Mixer1_Run )
   END_RUNG wire#w1
   RUNG wire#powerrail
      Contact( "Data".GlobalErrorStop )
   END_RUNG wire#w2
   RUNG wire#powerrail
      I_Contact( "Di_Ga1.4" )
   END_RUNG wire#w2
   // the same network as SCL:
   "Mixer1_Work_DB"(Start := "Data".Mixer1_Run,   // "MixerWork"
                    PowerIn := "Data".Mixer1.Power,
                    RegimBothSide := "Data".Mixer1.RegimBothSide,
                    TimeRight := "Data".Mixer1.TimeRight,
                    TimeLeft := "Data".Mixer1.TimeLeft,
                    TimePause := "Data".Mixer1.TimePause,
                    AvariyStop := "Data".GlobalErrorStop OR NOT "Di_Ga1.4");
END_REGION

REGION Network 9 (SCL): Показываем стрелки на визуализации 0 - нет стрелки, 1 - вправо, 2 - влево
   IF NOT "DrvCell_M1_1".Km1 THEN
       "Data".Mixer1.Direction := 0;
   ELSIF "DrvCell_M1_1".Km1 AND "DriveM1_1".Vx >= 2.0 THEN
       "Data".Mixer1.Direction := 1;
   ELSIF "DrvCell_M1_1".Km1 AND "DriveM1_1".Vx <= -2.0 THEN
       "Data".Mixer1.Direction := 2;
   END_IF;
END_REGION
END_FUNCTION

FUNCTION "Kristalizer2_Work" : Void   // FC12, LAD
{ S7_Optimized_Access := 'TRUE' }
VERSION : 0.1
   VAR_TEMP   // added for the SCL form of the ladder/FBD networks
      _w1 : Bool;
      _w2 : Bool;
      _w3 : Bool;
   END_VAR
BEGIN

REGION Network 1: Готовность маршрута
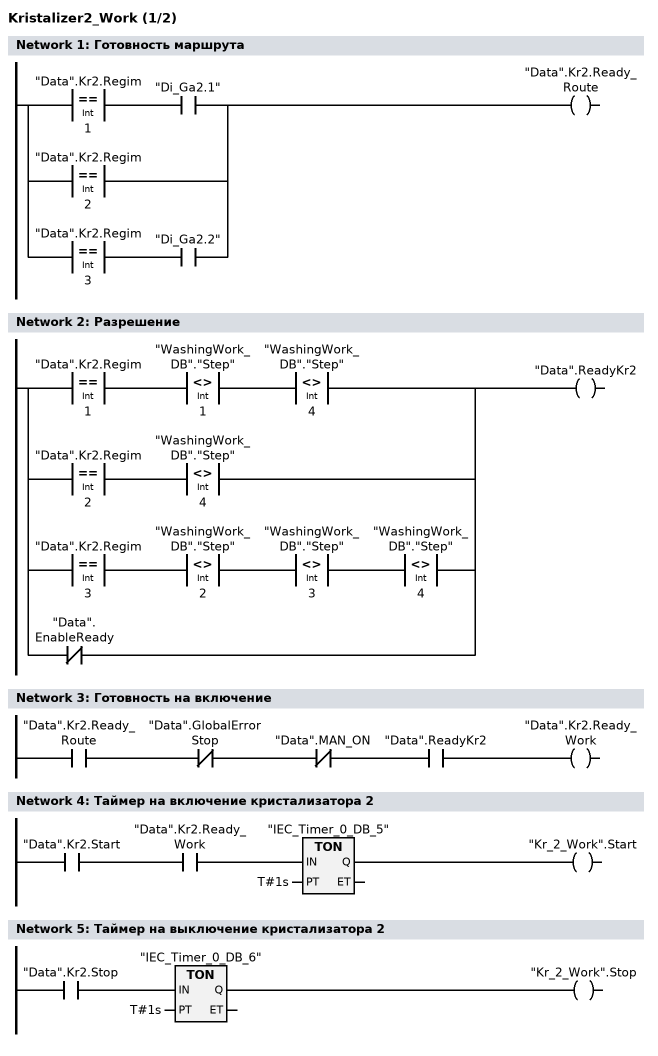
   RUNG wire#powerrail
      { S7_Templates := "SrcType := Int" } EQ_Contact(in1 := "Data".Kr2.Regim, in2 := 1)
      Contact( "Di_Ga2.1" )
      wire#w1
      Coil( "Data".Kr2.Ready_Route )
   END_RUNG
   RUNG wire#powerrail
      { S7_Templates := "SrcType := Int" } EQ_Contact(in1 := "Data".Kr2.Regim, in2 := 2)
   END_RUNG wire#w1
   RUNG wire#powerrail
      { S7_Templates := "SrcType := Int" } EQ_Contact(in1 := "Data".Kr2.Regim, in2 := 3)
      Contact( "Di_Ga2.2" )
   END_RUNG wire#w1
   // the same network as SCL:
   "Data".Kr2.Ready_Route := (("Data".Kr2.Regim = 1) AND "Di_Ga2.1") OR ("Data".Kr2.Regim = 2) OR (("Data".Kr2.Regim = 3) AND "Di_Ga2.2");
END_REGION

REGION Network 2: Разрешение
   RUNG wire#powerrail
      { S7_Templates := "SrcType := Int" } EQ_Contact(in1 := "Data".Kr2.Regim, in2 := 1)
      { S7_Templates := "SrcType := Int" } NE_Contact(in1 := "WashingWork_DB"."Step", in2 := 1)
      { S7_Templates := "SrcType := Int" } NE_Contact(in1 := "WashingWork_DB"."Step", in2 := 4)
      wire#w1
      Coil( "Data".ReadyKr2 )
   END_RUNG
   RUNG wire#powerrail
      { S7_Templates := "SrcType := Int" } EQ_Contact(in1 := "Data".Kr2.Regim, in2 := 2)
      { S7_Templates := "SrcType := Int" } NE_Contact(in1 := "WashingWork_DB"."Step", in2 := 4)
   END_RUNG wire#w1
   RUNG wire#powerrail
      { S7_Templates := "SrcType := Int" } EQ_Contact(in1 := "Data".Kr2.Regim, in2 := 3)
      { S7_Templates := "SrcType := Int" } NE_Contact(in1 := "WashingWork_DB"."Step", in2 := 2)
      { S7_Templates := "SrcType := Int" } NE_Contact(in1 := "WashingWork_DB"."Step", in2 := 3)
      { S7_Templates := "SrcType := Int" } NE_Contact(in1 := "WashingWork_DB"."Step", in2 := 4)
   END_RUNG wire#w1
   RUNG wire#powerrail
      I_Contact( "Data".EnableReady )
   END_RUNG wire#w1
   // the same network as SCL:
   "Data".ReadyKr2 := (("Data".Kr2.Regim = 1) AND ("WashingWork_DB"."Step" <> 1) AND ("WashingWork_DB"."Step" <> 4)) OR (("Data".Kr2.Regim = 2) AND ("WashingWork_DB"."Step" <> 4)) OR (("Data".Kr2.Regim = 3) AND ("WashingWork_DB"."Step" <> 2) AND ("WashingWork_DB"."Step" <> 3) AND ("WashingWork_DB"."Step" <> 4)) OR NOT "Data".EnableReady;
END_REGION

REGION Network 3: Готовность на включение
   RUNG wire#powerrail
      Contact( "Data".Kr2.Ready_Route )
      I_Contact( "Data".GlobalErrorStop )
      I_Contact( "Data".MAN_ON )
      Contact( "Data".ReadyKr2 )
      Coil( "Data".Kr2.Ready_Work )
   END_RUNG
   // the same network as SCL:
   "Data".Kr2.Ready_Work := "Data".Kr2.Ready_Route AND NOT "Data".GlobalErrorStop AND NOT "Data".MAN_ON AND "Data".ReadyKr2;
END_REGION

REGION Network 4: Таймер на включение кристализатора 2
   "IEC_Timer_0_DB_5".TON(IN := "Data".Kr2.Start AND "Data".Kr2.Ready_Work, PT := T#1s);
   "Kr_2_Work".Start := "IEC_Timer_0_DB_5".Q;
END_REGION

REGION Network 5: Таймер на выключение кристализатора 2
   "IEC_Timer_0_DB_6".TON(IN := "Data".Kr2.Stop, PT := T#1s);
   "Kr_2_Work".Stop := "IEC_Timer_0_DB_6".Q;
END_REGION

REGION Network 6: Работа кристализатора №2
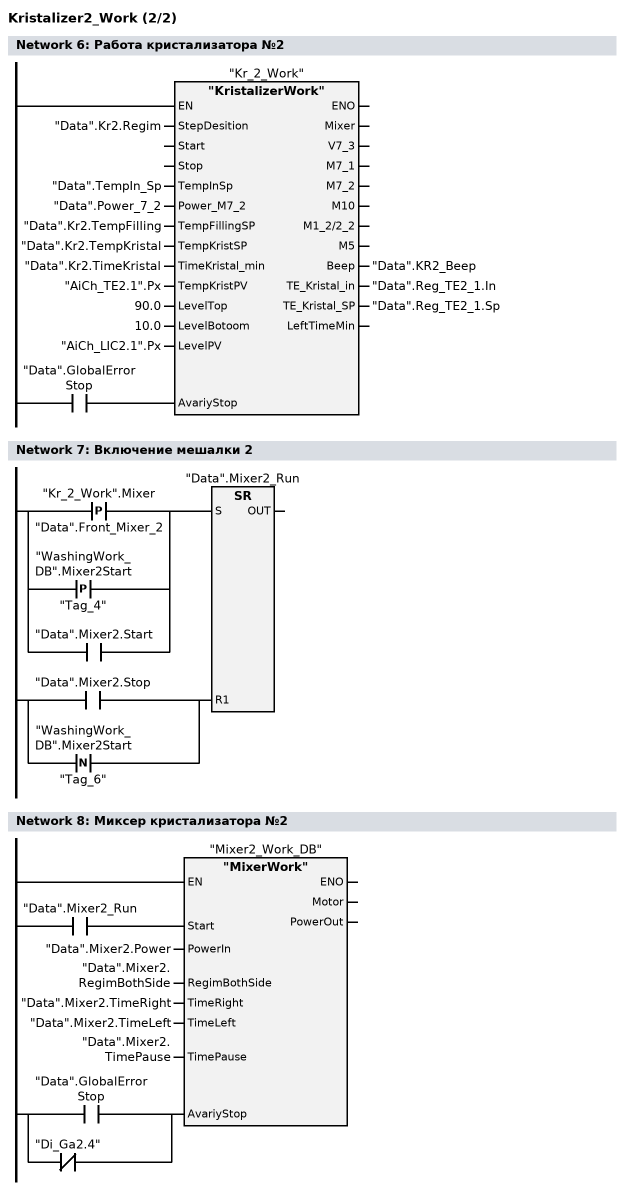
   RUNG wire#powerrail
      "Kr_2_Work"(AvariyStop := wire#w1, StepDesition := "Data".Kr2.Regim, Start :=, Stop :=, TempInSp := "Data".TempIn_Sp, Power_M7_2 := "Data".Power_7_2, TempFillingSP := "Data".Kr2.TempFilling, TempKristSP := "Data".Kr2.TempKristal, TimeKristal_min := "Data".Kr2.TimeKristal, TempKristPV := "AiCh_TE2.1".Px, LevelTop := 90.0, LevelBotoom := 10.0, LevelPV := "AiCh_LIC2.1".Px, Mixer =>, V7_3 =>, M7_1 =>, M7_2 =>, M10 =>, "M1_2/2_2" =>, M5 =>, Beep => "Data".KR2_Beep, TE_Kristal_in => "Data".Reg_TE2_1.In, TE_Kristal_SP => "Data".Reg_TE2_1.Sp, LeftTimeMin =>)
   END_RUNG
   RUNG wire#powerrail
      Contact( "Data".GlobalErrorStop )
   END_RUNG wire#w1
   // the same network as SCL:
   "Kr_2_Work"(StepDesition := "Data".Kr2.Regim,   // "KristalizerWork"
               TempInSp := "Data".TempIn_Sp,
               Power_M7_2 := "Data".Power_7_2,
               TempFillingSP := "Data".Kr2.TempFilling,
               TempKristSP := "Data".Kr2.TempKristal,
               TimeKristal_min := "Data".Kr2.TimeKristal,
               TempKristPV := "AiCh_TE2.1".Px,
               LevelTop := 90.0,
               LevelBotoom := 10.0,
               LevelPV := "AiCh_LIC2.1".Px,
               AvariyStop := "Data".GlobalErrorStop,
               Beep => "Data".KR2_Beep,
               TE_Kristal_in => "Data".Reg_TE2_1.In,
               TE_Kristal_SP => "Data".Reg_TE2_1.Sp);
END_REGION

REGION Network 7: Включение мешалки 2
   RUNG wire#powerrail
      P_Contact(operand := "Kr_2_Work".Mixer, bit := "Data".Front_Mixer_2)
      wire#w1
      S_SR(operand := "Data".Mixer2_Run, r1 := wire#w2)
   END_RUNG
   RUNG wire#powerrail
      P_Contact(operand := "WashingWork_DB".Mixer2Start, bit := "Tag_4")
   END_RUNG wire#w1
   RUNG wire#powerrail
      Contact( "Data".Mixer2.Start )
   END_RUNG wire#w1
   RUNG wire#powerrail
      Contact( "Data".Mixer2.Stop )
   END_RUNG wire#w2
   RUNG wire#powerrail
      N_Contact(operand := "WashingWork_DB".Mixer2Start, bit := "Tag_6")
   END_RUNG wire#w2
   // the same network as SCL:
   #_w1 := "Kr_2_Work".Mixer AND NOT "Data".Front_Mixer_2;   // rising edge of "Kr_2_Work".Mixer
   "Data".Front_Mixer_2 := "Kr_2_Work".Mixer;
   #_w2 := "WashingWork_DB".Mixer2Start AND NOT "Tag_4";   // rising edge of "WashingWork_DB".Mixer2Start
   "Tag_4" := "WashingWork_DB".Mixer2Start;
   #_w3 := NOT "WashingWork_DB".Mixer2Start AND "Tag_6";   // falling edge of "WashingWork_DB".Mixer2Start
   "Tag_6" := "WashingWork_DB".Mixer2Start;
   IF #_w1 OR #_w2 OR "Data".Mixer2.Start THEN
       "Data".Mixer2_Run := TRUE;   // SR flip-flop
   END_IF;
   IF "Data".Mixer2.Stop OR #_w3 THEN "Data".Mixer2_Run := FALSE; END_IF;
END_REGION

REGION Network 8: Миксер кристализатора №2
   RUNG wire#powerrail
      "Mixer2_Work_DB"(Start := wire#w1, AvariyStop := wire#w2, PowerIn := "Data".Mixer2.Power, RegimBothSide := "Data".Mixer2.RegimBothSide, TimeRight := "Data".Mixer2.TimeRight, TimeLeft := "Data".Mixer2.TimeLeft, TimePause := "Data".Mixer2.TimePause, Motor =>, PowerOut =>)
   END_RUNG
   RUNG wire#powerrail
      Contact( "Data".Mixer2_Run )
   END_RUNG wire#w1
   RUNG wire#powerrail
      Contact( "Data".GlobalErrorStop )
   END_RUNG wire#w2
   RUNG wire#powerrail
      I_Contact( "Di_Ga2.4" )
   END_RUNG wire#w2
   // the same network as SCL:
   "Mixer2_Work_DB"(Start := "Data".Mixer2_Run,   // "MixerWork"
                    PowerIn := "Data".Mixer2.Power,
                    RegimBothSide := "Data".Mixer2.RegimBothSide,
                    TimeRight := "Data".Mixer2.TimeRight,
                    TimeLeft := "Data".Mixer2.TimeLeft,
                    TimePause := "Data".Mixer2.TimePause,
                    AvariyStop := "Data".GlobalErrorStop OR NOT "Di_Ga2.4");
END_REGION

REGION Network 9 (SCL): Показываем стрелки на визуализации 0 - нет стрелки, 1 - вправо, 2 - влево
   IF NOT "DrvCell_M2_1".Km1 THEN
       "Data".Mixer2.Direction := 0;
   ELSIF "DrvCell_M2_1".Km1 AND "DriveM2_1".Vx >= 2.0 THEN
       "Data".Mixer2.Direction := 1;
   ELSIF "DrvCell_M2_1".Km1 AND "DriveM2_1".Vx <= -2.0 THEN
       "Data".Mixer2.Direction := 2;
   END_IF;
END_REGION
END_FUNCTION

// folder: Lines

FUNCTION_BLOCK "ViewLine"   // FB9, SCL
{ S7_Optimized_Access := 'TRUE' }
VERSION : 0.1
   VAR_OUTPUT
      Line1 : Int;
      Line2 : Int;
      Line3 : Int;
      Line4 : Int;
      Line5 : Int;
      Line6 : Int;
      Line7 : Int;
      Line8 : Int;
      Line9 : Int;
      Line10 : Int;
      Line11 : Int;
      Line12 : Int;
      Line13 : Int;
      Line14 : Int;
      Line15 : Int;
      Line16 : Int;
      Line17 : Int;
      Line18 : Int;
      Line19 : Int;
      Line20 : Int;
      Line21 : Int;
      Line22 : Int;
      Line23 : Int;
      Line24 : Int;
      Line25 : Int;
      Line26 : Int;
   END_VAR
BEGIN
   // Линия 1

   IF ("Kr_1_Work".Run OR "Kr_2_Work".Run) AND "DrvCell_V7_3".Km1 THEN
       #Line1 := 1;
   ELSIF "WashingWork_DB".Run AND "DrvCell_V7_3".Km1 THEN
       #Line1 := 2;
   ELSE
       #Line1 := 0;
   END_IF;


   // Линия 2
   IF ("Kr_1_Work".Run OR "Kr_2_Work".Run) AND "DrvCell_V7_4".Km1 THEN
       #Line2 := 1;
   ELSIF "WashingWork_DB".Run AND "DrvCell_V7_4".Km1 THEN
       #Line2 := 2;
   ELSE
       #Line2 := 0;
   END_IF;


   // Линия 3
   IF ("Kr_1_Work".Run OR "Kr_2_Work".Run) AND "DrvCell_M7_1".Km1 THEN
       #Line3 := 1;
   ELSIF "WashingWork_DB".Run AND "DrvCell_M7_1".Km1 THEN
       #Line3 := 2;
   ELSE
       #Line3 := 0;
   END_IF;


   // Линия 4
   IF ("Kr_1_Work".Run OR "Kr_2_Work".Run) AND "DrvCell_M7_2".Km1 THEN
       #Line4 := 1;
   ELSIF "WashingWork_DB".Run AND "DrvCell_M7_2".Km1 THEN
       #Line4 := 2;
   ELSE
       #Line4 := 0;
   END_IF;


   // Линия 5
   IF ("Kr_1_Work".Run OR "Kr_2_Work".Run) AND "DrvCell_M10".Km1 THEN
       #Line5 := 1;
   ELSIF "WashingWork_DB".Run AND "DrvCell_M10".Km1 THEN
       #Line5 := 2;
   ELSE
       #Line5 := 0;
   END_IF;

   // Линия 6
   IF ("Kr_1_Work".Run OR "Kr_2_Work".Run) AND NOT "Data".GlobalErrorStop THEN
       #Line6 := 1;
   ELSIF "WashingWork_DB".Run AND NOT "Data".GlobalErrorStop THEN
       #Line6 := 2;
   ELSE
       #Line6 := 0;
   END_IF;

   // Линия 7
   IF ("Kr_1_Work".Run OR "Kr_2_Work".Run) AND "Data".Reg_01RV01.LMN >= 2.0 THEN
       #Line7 := 1;
   ELSIF "WashingWork_DB".Run AND "Data".Reg_01RV01.LMN >= 2.0 THEN
       #Line7 := 2;
   ELSE
       #Line7 := 0;
   END_IF;

   // Линия 8
   IF ("Kr_1_Work".Run OR "Kr_2_Work".Run) AND "DrvCell_M7_1".Km1 THEN
       #Line8 := 1;
   ELSIF "WashingWork_DB".Run AND "DrvCell_M7_1".Km1 THEN
       #Line8 := 2;
   ELSE
       #Line8 := 0;
   END_IF;

   // Линия 9
   IF ("Kr_1_Work".Run OR "Kr_2_Work".Run) AND "DrvCell_M7_2".Km1 THEN
       #Line9 := 1;
   ELSIF "WashingWork_DB".Run AND "DrvCell_M7_2".Km1 THEN
       #Line9 := 2;
   ELSE
       #Line9 := 0;
   END_IF;

   // Линия 10 - 1 кристализатор-----------------------------------------------------
   IF ("Kr_1_Work"."Step" = 1 AND "DrvCell_M7_1".Km1) OR ("Kr_1_Work"."Step" = 3 AND "DrvCell_M5".Km1) THEN
       #Line10 := 1;
   ELSIF "WashingWork_DB"."Step" = 3 AND  "DrvCell_M4".Km1 THEN
       #Line10 := 2;
   ELSE
       #Line10 := 0;
   END_IF;

   // Линия 11
   IF "Data".Equipment_Work AND"DrvCell_M1_2".Km1 THEN
       #Line11 := 1;
   ELSE
       #Line11 := 0;
   END_IF;

   // Линия 12
   IF "Data".Equipment_Work AND "DrvCell_V1_1".Km1 THEN
       #Line12 := 1;
   ELSE
       #Line12 := 0;
   END_IF;

   // Линия 13
   IF "Data".Equipment_Work AND "DrvCell_V1_7".Km1 THEN
       #Line13 := 1;
   ELSE
       #Line13 := 0;
   END_IF;

   // Линия 14 - 2 кристализатор-----------------------------------------------------
   IF ("Kr_2_Work"."Step" = 1 AND "DrvCell_M7_1".Km1) OR ("Kr_2_Work"."Step" = 3 AND "DrvCell_M5".Km1) THEN
       #Line14 := 1;
   ELSIF "WashingWork_DB"."Step" = 4 AND "DrvCell_M4".Km1 THEN
       #Line14 := 2;
   ELSE
       #Line14 := 0;
   END_IF;

   // Линия 15
   IF "Data".Equipment_Work AND "DrvCell_M2_2".Km1 THEN
       #Line15 := 1;
   ELSE
       #Line15 := 0;
   END_IF;

   // Линия 16
   IF "Data".Equipment_Work AND "DrvCell_V2_1".Km1 THEN
       #Line16 := 1;
   ELSE
       #Line16 := 0;
   END_IF;

   // Линия 17
   IF "Data".Equipment_Work AND "DrvCell_V2_7".Km1 THEN
       #Line17 := 1;
   ELSE
       #Line17 := 0;
   END_IF;

   // Линия 18
   IF "Kr_1_Work"."Step" = 3 THEN
       #Line18 := 1;
   ELSIF ("WashingWork_DB"."Step" = 2 OR "WashingWork_DB"."Step" = 3) AND "DrvCell_M4".Km1 THEN 
       #Line18 := 2;
   ELSE
       #Line18 := 0;
   END_IF;

   // Линия 19
   IF ("Kr_1_Work"."Step" = 3 OR "Kr_2_Work"."Step" = 3) AND "DrvCell_M5".Km1 THEN
       #Line19 := 1;
   ELSIF ("WashingWork_DB"."Step" = 2 OR "WashingWork_DB"."Step" = 3 OR "WashingWork_DB"."Step" = 4) AND "DrvCell_M4".Km1 THEN
       #Line19 := 2;
   ELSE
       #Line19 := 0;
   END_IF;

   // Линия 20
   IF ("Kr_1_Work"."Step" = 3 OR "Kr_2_Work"."Step" = 3) AND "DrvCell_M5".Km1 THEN
       #Line20 := 1;
   ELSIF ("WashingWork_DB"."Step" = 2 OR "WashingWork_DB"."Step" = 3 OR "WashingWork_DB"."Step" = 4) AND "DrvCell_M5".Km1 THEN
       #Line20 := 2;
   ELSE
       #Line20 := 0;
   END_IF;

   // Линия 21
   IF ("WashingWork_DB"."Step" = 2 OR "WashingWork_DB"."Step" = 3 OR "WashingWork_DB"."Step" = 4) AND "DrvCell_M5".Km1 THEN
       #Line21 := 1;
   ELSE
       #Line21 := 0;
   END_IF;

   // Линия 22
   IF ("WashingWork_DB"."Step" = 2 OR "WashingWork_DB"."Step" = 3 OR "WashingWork_DB"."Step" = 4) AND "DrvCell_M4".Km1 THEN
       #Line22 := 1;
   ELSE
       #Line22 := 0;
   END_IF;

   // Линия 23
   IF "WashingWork_DB"."Step" = 2 AND "DrvCell_M4".Km1 THEN
       #Line23 := 1;
   ELSE
       #Line23 := 0;
   END_IF;


   // Линия 24
   IF "WashingWork_DB"."Step" = 3 AND "DrvCell_M4".Km1 THEN
       #Line24 := 1;
   ELSE
       #Line24 := 0;
   END_IF;

   // Линия 25
   IF "WashingWork_DB"."Step" = 4 AND "DrvCell_M4".Km1 THEN
       #Line25 := 1;
   ELSE
       #Line25 := 0;
   END_IF;
END_FUNCTION_BLOCK

FUNCTION "LinesFC" : Void   // FC1, LAD
{ S7_Optimized_Access := 'TRUE' }
VERSION : 0.1
BEGIN

REGION Network 1
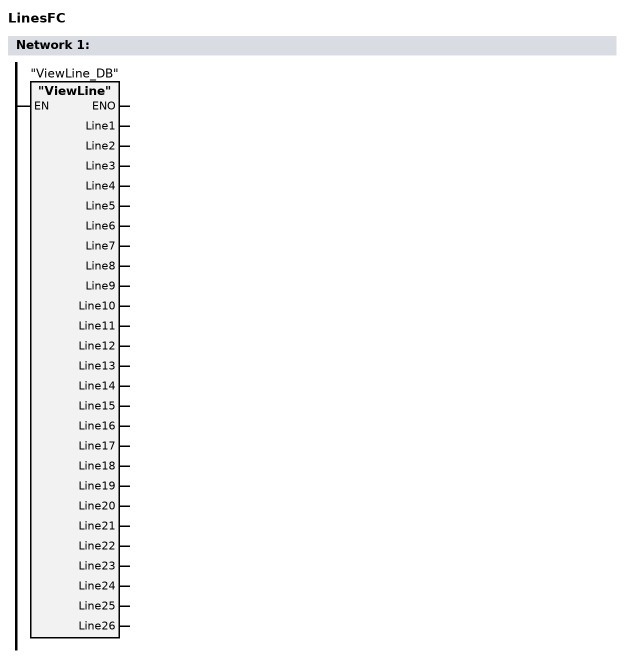
   RUNG wire#powerrail
      "ViewLine_DB"(Line1 =>, Line2 =>, Line3 =>, Line4 =>, Line5 =>, Line6 =>, Line7 =>, Line8 =>, Line9 =>, Line10 =>, Line11 =>, Line12 =>, Line13 =>, Line14 =>, Line15 =>, Line16 =>, Line17 =>, Line18 =>, Line19 =>, Line20 =>, Line21 =>, Line22 =>, Line23 =>, Line24 =>, Line25 =>, Line26 =>)
   END_RUNG
   // the same network as SCL:
   "ViewLine_DB"();   // "ViewLine"
END_REGION
END_FUNCTION

// folder: Messages

FUNCTION "Messag" : Void   // FC5, SCL
{ S7_Optimized_Access := 'TRUE' }
VERSION : 0.1
BEGIN
   "Messages".Message1 := "FpDW_DB".F[34]; // Нажат аварийный стоп
   "Messages".Message2 := "FpDW_DB".F[35]; // Напряжение 380 вольт не внорме
   "Messages".Message3 := "FpDW_DB".F[36]; // Давление воздуха
   "Messages".Message4 := "FpDW_DB".F[37]; // верхний уровень кристализатора 1
   "Messages".Message5 := "FpDW_DB".F[38]; // верхний уровень кристализатора 2
   "Messages".Message6 := "FpDW_DB".F[39]; // 


   // Warnings--------------------------------------------------------

   "Messages".Message7 := "Di_BatRaz"; // батарея разряжена
   "Messages".Message8 := "Di_BatFault"; // батарея неисправна
   "Messages".Message9 := "FpDW_DB".F[40]; // Открыт люк 1 кристализатора
   "Messages".Message10 := "FpDW_DB".F[41]; // Открыт люк 2 кристализатора
END_FUNCTION

// folder: Pumps&Valves

FUNCTION "Pumps&Valves" : Void   // FC7, SCL
{ S7_Optimized_Access := 'TRUE' }
VERSION : 0.1
BEGIN
   // Насос M1_1
   "DrvCell_M1_1"(QFx := "Di_Qf1.1",
                  Flt := "DriveM1_1".Flt,
                  Mdx := NOT "Data".MAN_ON,
                  Kb_Sr1:=1,
                  Cm1 := "Mixer1_Work_DB".Motor AND NOT "DrvCell_M1_1".Err,
                  Km1 => "DriveM1_1".Run);

   // Насос M1_2
   "DrvCell_M1_2"(Kx1 := "Di_Km1.2",
                  Mdx := NOT "Data".MAN_ON,
                  Cm1 := "Kr_1_Work"."M1_2/2_2" AND NOT "DrvCell_M1_2".Err,
                  Kb_Sr1 := 1,
                  Md_Kx1 := 1,
                  Md_TmX := T#5S,
                  Md_TmD := T#5S,
                  Km1 => "Dq_Km1.2");

   // Насос M2_1
   "DrvCell_M2_1"(QFx := "Di_Qf2.1",
                  Flt := "DriveM2_1".Flt,
                  Mdx := NOT "Data".MAN_ON,
                  Cm1 := "Mixer2_Work_DB".Motor AND NOT "DrvCell_M2_1".Err,
                  Kb_Sr1 := 1,
                  Km1 => "DriveM2_1".Run);

   // Насос M2_2
   "DrvCell_M2_2"(Kx1 := "Di_Km2.2",
                  Mdx := NOT "Data".MAN_ON,
                  Cm1 := "Kr_2_Work"."M1_2/2_2" AND NOT "DrvCell_M2_2".Err,
                  Kb_Sr1 := 1,
                  Md_Kx1 := 1,
                  Md_TmX := T#5S,
                  Md_TmD := T#5S,
                  Km1 => "Dq_Km2.2");

   // Насос 3
   "DrvCell_M3"(Kx1:="Di_Km03",
                   Mdx:=NOT "Data".MAN_ON,
                   Cm1:="IceWaterWork_DB".M3 AND NOT "DrvCell_M3".Err,
                   Kb_Sr1:=1,
                   Md_Kx1:=1,
                   Md_TmX:=T#5S,
                   Md_TmD:=T#5S,
                   Km1=>"Dq_Km3");


   // Насос 4
   "DrvCell_M4"(Kx1 := "Di_Km04",
                Mdx := NOT "Data".MAN_ON,
                Cm1 :=  "WashingWork_DB".M4 AND NOT "DrvCell_M4".Err,
                Kb_Sr1 := 1,
                Md_Kx1 := 1,
                Md_TmX := T#5S,
                Md_TmD := T#5S,
                Km1 => "Dq_Km4");

   // Насос 5
   "DrvCell_M5"(Mdx := NOT "Data".MAN_ON,
                Cm1 := ("Kr_1_Work".M5 OR "Kr_2_Work".M5 OR "WashingWork_DB".M5) AND NOT "DrvCell_M5".Err,
                Kb_Sr1 := 1);

   // Насос 7_1
   "DrvCell_M7_1"(QFx := "Di_QF7.1",
                  Flt := "DriveM7_1".Flt,
                  Mdx := NOT "Data".MAN_ON,
                  Cm1 := ("Kr_1_Work".M7_1 OR "Kr_2_Work".M7_1 OR "WashingWork_DB".M7_1) AND NOT "DrvCell_M7_1".Err ,
                  Kb_Sr1 := 1,
                  Km1 => "DriveM7_1".Run);

   // Насос 7_2
   "DrvCell_M7_2"(QFx := "Di_QF7.2",
                  Flt := "DriveM7_2".Flt,
                  Mdx := NOT "Data".MAN_ON,
                  Cm1 := ("Kr_1_Work".M7_2 OR "Kr_2_Work".M7_2 OR "WashingWork_DB".M7_2) AND NOT "DrvCell_M7_2".Err ,
                  Kb_Sr1 := 1,
                  Km1 => "DriveM7_2".Run);

   // Насос 10
   "DrvCell_M10"(Mdx:=NOT "Data".MAN_ON,
                 Kx1:="Di_Km10",
                 Cm1:=("Kr_1_Work".M10 OR "Kr_2_Work".M10) AND NOT "DrvCell_M10".Err,
                 Kb_Sr1:=1,
                 Md_Kx1:=1,
                 Md_TmX:=T#5S,
                 Md_TmD:=T#5S,
                 Km1=>"Dq_Km10"
                 );

   //------------------------------------------ Клапана------------------------------------
   // Клапан 7.1
   "DrvCell_V7_1"(Mdx:=NOT "Data".MAN_ON,
                  Cm1:="DrvCell_M7_1".Km1 AND NOT "DrvCell_V7_1".Err,
                  Kb_Sr1:=1,
                  Km1=>"Dq_V7.1");

   // Клапан 7.2
   "DrvCell_V7_2"(Mdx:=NOT "Data".MAN_ON,
                  Cm1:="DrvCell_M7_2".Km1 AND NOT "DrvCell_V7_2".Err,
                  Kb_Sr1:=1,
                  Km1=>"Dq_V7.2");

   // Клапан 1.1
   "DrvCell_V1_1"(Mdx:=NOT "Data".MAN_ON,
                  Cm1:="Data".Reg_TE1_1.V1_1 AND NOT "DrvCell_V1_1".Err,
                  Kb_Sr1:=1,
                  Km1=>"Dq_V1.1");

   // Клапан 2.1
   "DrvCell_V2_1"(Mdx:=NOT "Data".MAN_ON,
                   Cm1:="Data".Reg_TE2_1.V2_1 AND NOT "DrvCell_V2_1".Err,
                   Kb_Sr1:=1,
                   Km1=>"Dq_V2.1");

    // Клапан 3.1
    "DrvCell_V3_1"(Mdx:=NOT "Data".MAN_ON,
                   Kb_Sr1:=1,
                   Km1=>"Dq_V3.1");

    // Клапан 1.7
    "DrvCell_V1_7"(Mdx:=0,
                   Kb_Sb1:=1,
                   Km1=>"Dq_V1.7"
                   );

    // Клапан 2.7
    "DrvCell_V2_7"(Mdx:=0,
                   Kb_Sb1:=1,
                   Km1=>"Dq_V2.7");

    // Клапан 3.7
    "DrvCell_V3_7"(Mdx:=NOT "Data".MAN_ON,
                   Kb_Sr1:=1,
                   Km1=>"Dq_V3.7");

    // Клапан 7.3
    "DrvCell_V7_3"( Mdx:=NOT "Data".MAN_ON,
                   Cm1:=("Kr_1_Work".V7_3 OR "Kr_2_Work".V7_3 OR "WashingWork_DB".V7_3) AND NOT "DrvCell_V7_3".Err,
                   Kb_Sr1:=1,
                   Km1=>"Dq_V7.3");

    // Клапан 7.4
    "DrvCell_V7_4"(Mdx:=NOT "Data".MAN_ON,
                   Cm1:="WashingWork_DB".V7_4 AND NOT "DrvCell_V7_4".Err,
                   Kb_Sr1:=1,
                   Km1=>"Dq_V7.4");

    // Аварийный звонок 
    IF "Data".Erorrs_Beep OR "Data".KR1_Beep OR "Data".KR2_Beep THEN
        "Dq_KB1" := TRUE;
    ELSE
        "Dq_KB1" := FALSE;
    END_IF;
END_FUNCTION

// folder: RegPID

FUNCTION "REG_PID" : Void   // FC6, LAD
{ S7_Optimized_Access := 'TRUE' }
VERSION : 0.1
BEGIN

REGION Network 1: 1RV01
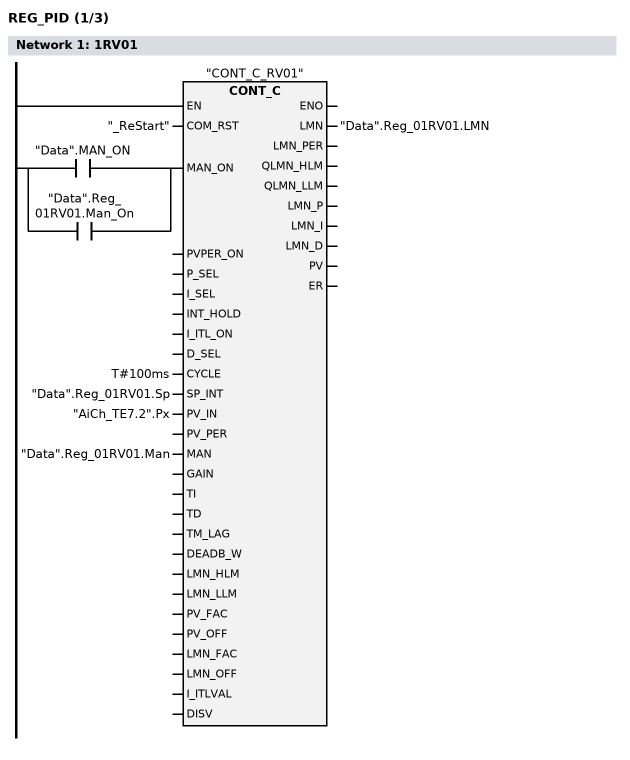
   "CONT_C_RV01"(COM_RST := "_ReStart",   // CONT_C
                 MAN_ON := "Data".MAN_ON OR "Data".Reg_01RV01.Man_On,
                 CYCLE := T#100ms,
                 SP_INT := "Data".Reg_01RV01.Sp,
                 PV_IN := "AiCh_TE7.2".Px,
                 MAN := "Data".Reg_01RV01.Man,
                 LMN => "Data".Reg_01RV01.LMN);
END_REGION

REGION Network 2: M7_1
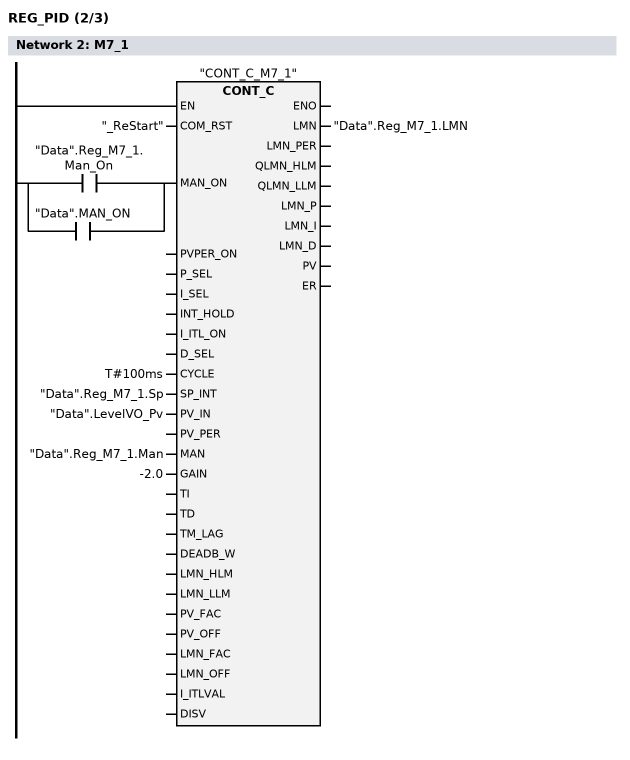
   "CONT_C_M7_1"(COM_RST := "_ReStart",   // CONT_C
                 MAN_ON := "Data".Reg_M7_1.Man_On OR "Data".MAN_ON,
                 CYCLE := T#100ms,
                 SP_INT := "Data".Reg_M7_1.Sp,
                 PV_IN := "Data".LevelVO_Pv,
                 MAN := "Data".Reg_M7_1.Man,
                 GAIN := -2.0,
                 LMN => "Data".Reg_M7_1.LMN);
END_REGION

REGION Network 3: M7_2
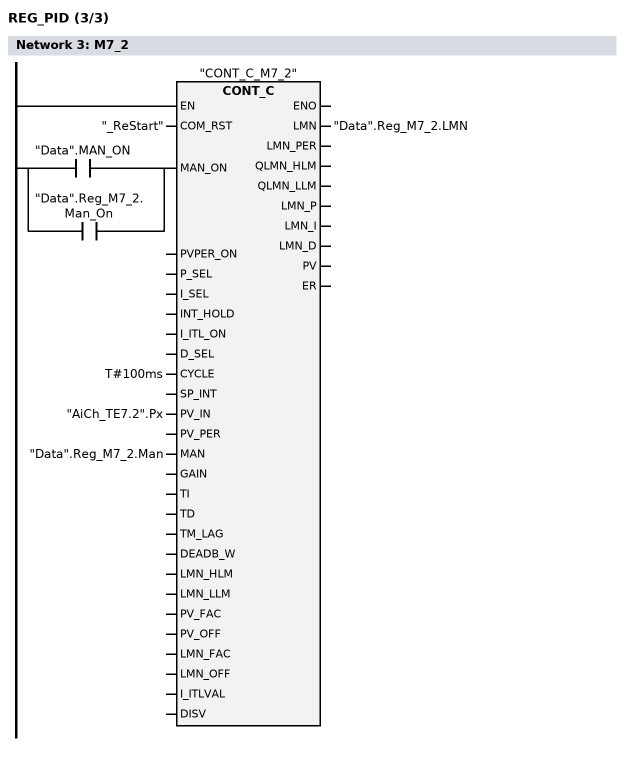
   "CONT_C_M7_2"(COM_RST := "_ReStart",   // CONT_C
                 MAN_ON := "Data".MAN_ON OR "Data".Reg_M7_2.Man_On,
                 CYCLE := T#100ms,
                 PV_IN := "AiCh_TE7.2".Px,
                 MAN := "Data".Reg_M7_2.Man,
                 LMN => "Data".Reg_M7_2.LMN);
END_REGION

REGION Network 4 (SCL): Регулятор температуры TE1.1 в кристализаторе №1
   IF "Data".Reg_TE1_1.In THEN
       IF ("AiCh_TE1.1".Px >= "Data".Reg_TE1_1.Sp + "Data".Reg_TE1_1.Gis) THEN
           "Data".Reg_TE1_1.V1_1 := TRUE;
       END_IF;
       IF ("AiCh_TE1.1".Px <= "Data".Reg_TE1_1.Sp - "Data".Reg_TE1_1.Gis) THEN
           "Data".Reg_TE1_1.V1_1 := FALSE;
       END_IF;
   ELSE
       "Data".Reg_TE1_1.V1_1 := FALSE;
   END_IF;
END_REGION

REGION Network 5 (SCL): Регулятор температуры TE2.1 в кристализаторе №1
   IF "Data".Reg_TE2_1.In THEN
       IF ("AiCh_TE2.1".Px >= "Data".Reg_TE2_1.Sp + "Data".Reg_TE2_1.Gis) THEN
           "Data".Reg_TE2_1.V2_1 := TRUE;
       END_IF;
       IF ("AiCh_TE2.1".Px <= "Data".Reg_TE2_1.Sp - "Data".Reg_TE2_1.Gis) THEN
           "Data".Reg_TE2_1.V2_1 := FALSE;
       END_IF;
   ELSE
       "Data".Reg_TE2_1.V2_1 := FALSE;
   END_IF;
END_REGION
END_FUNCTION

// folder: Sys

FUNCTION_BLOCK "Sys"   // FB1, SCL
{ S7_Optimized_Access := 'TRUE' }
VERSION : 0.1
   VAR
      Tm : "SysTime";
      TmWork : DInt := 0;
      FmWork : Bool := 0;
   END_VAR
BEGIN
   // Формируем текущее циклическое системное время в MD20 (_TIME)
   #Tm();

   "_ReStart" := "_Start";
   IF ("_Start") THEN
       #TmWork := 0;
       #FmWork := 0;
       "_MEn" := 1;
   ELSIF (#TmWork < 100) THEN
       #TmWork := #TmWork + 1;
       IF (#TmWork = 95) THEN
           "_ACK" := 1;
       END_IF;
       IF (#TmWork = 98) THEN
           "_ACK" := 0;
       END_IF;
   END_IF;

   // Обще квитирование
   "_ACK" := "Di_ACK" OR "Data".Ack;

   "_HALT" := NOT "Di_AvarStop";

   // Передача времени на панель
    "Panel_AreaPointer".DateTimePLC.DateTime := #Tm.DTx;
END_FUNCTION_BLOCK

FUNCTION "REG_Zero" : Void   // FC11, SCL
{ S7_Optimized_Access := 'TRUE' }
VERSION : 0.1
BEGIN

   // Регулятор 01RV01
   "Data".Reg_01RV01.Man_On := TRUE;
   "Data".Reg_01RV01.Man := 0.0;

   // Регулятор M7_1
   "Data".Reg_M7_1.Man_On := TRUE;
   "Data".Reg_M7_1.Man := 0.0;

   // Регулятор M7_2
   "Data".Reg_M7_2.Man_On := TRUE;
   "Data".Reg_M7_2.Man := 0.0;

   // Частотник М1_1
   "Data".Mixer1.Man := 0;

   // Частотник М1_2
   "Data".Mixer2.Man := 0;
END_FUNCTION

// folder: Washing

FUNCTION_BLOCK "WashingWork"   // FB3, SCL
{ S7_Optimized_Access := 'TRUE' }
VERSION : 0.1
   VAR_INPUT
      StepDesition : Int := 1;
      Power_M7_2 : Real;
      Start : Bool;
      Stop : Bool;
      AvariyStop : Bool;
   END_VAR
   VAR_OUTPUT
      V7_3 : Bool;
      V7_4 : Bool;
      M7_1 : Bool;
      M7_2 : Bool;
      M5 : Bool;
      M4 : Bool;
      Mixer1Start : Bool;
      Mixer2Start : Bool;
   END_VAR
   VAR
      FrontStart : R_TRIG;
      FrontStop : R_TRIG;
      Run : Bool;
      Flip : "FlipSingle";
      "Step" : Int;
   END_VAR
BEGIN
   #Flip(Time_work := 60,
         Time_pause := 30);

   #FrontStart(CLK := #Start);
   #FrontStop(CLK := #Stop);

   IF #FrontStart.Q THEN
       #Run := TRUE;
       #"Step" := #StepDesition;
   END_IF;

   IF #FrontStop.Q THEN
       #Run := FALSE;
   END_IF;


   IF #Run AND NOT #AvariyStop THEN

       CASE #"Step" OF
           1: // Мойка линии наполнения
               #Flip.in := TRUE;

               #V7_3 := TRUE;
               #V7_4 := true AND #Flip.out;

               "Data".Reg_M7_1.Man_On := TRUE;
               "Data".Reg_M7_1.Man := 100.0;

               "Data".Reg_M7_2.Man_On := TRUE;
               "Data".Reg_M7_2.Man := #Power_M7_2;

               #M7_1 := TRUE;
               #M7_2 := TRUE;

           2: // Мойка линии выгрузки
               #M5 := TRUE;
               #M4 := TRUE;


           3: // Мойка 1 кристализатора
               #Mixer1Start := TRUE;
               #M5 := TRUE;
               #M4 := TRUE;


           4: // Мойка 2 кристализатора 
               #Mixer2Start := TRUE;
               #M5 := TRUE;
               #M4 := TRUE;

       END_CASE;

   ELSE
       #Flip.in := FALSE;
       #V7_3 := FALSE;
       #V7_4 := FALSE;
       #M7_1 := FALSE;
       #M7_2 := FALSE;
       #M5 := FALSE;
       #M4 := FALSE;
       #Mixer1Start := FALSE;
       #Mixer2Start := FALSE;

       IF NOT #AvariyStop OR NOT #Run THEN
           #"Step" := 0;
       END_IF;
   END_IF;
END_FUNCTION_BLOCK

FUNCTION "Washing" : Void   // FC8, LAD
{ S7_Optimized_Access := 'TRUE' }
VERSION : 0.1
BEGIN

REGION Network 1: Готовность маршрута мойки
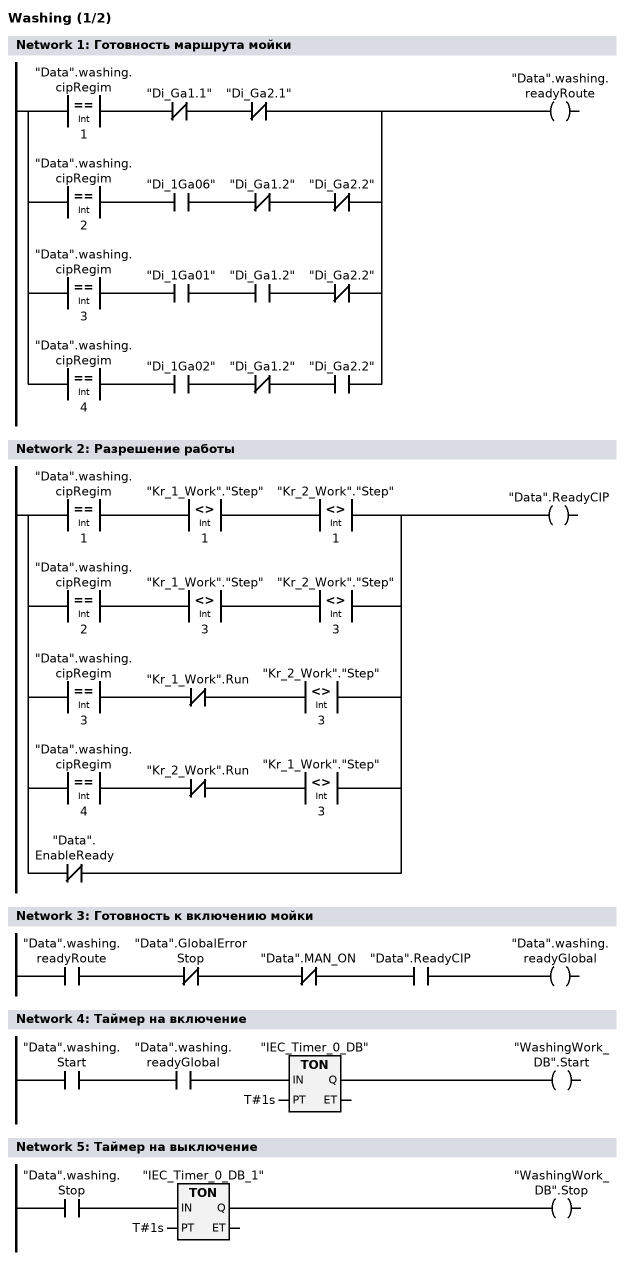
   RUNG wire#powerrail
      { S7_Templates := "SrcType := Int" } EQ_Contact(in1 := "Data".washing.cipRegim, in2 := 1)
      I_Contact( "Di_Ga1.1" )
      I_Contact( "Di_Ga2.1" )
      wire#w1
      Coil( "Data".washing.readyRoute )
   END_RUNG
   RUNG wire#powerrail
      { S7_Templates := "SrcType := Int" } EQ_Contact(in1 := "Data".washing.cipRegim, in2 := 2)
      Contact( "Di_1Ga06" )
      I_Contact( "Di_Ga1.2" )
      I_Contact( "Di_Ga2.2" )
   END_RUNG wire#w1
   RUNG wire#powerrail
      { S7_Templates := "SrcType := Int" } EQ_Contact(in1 := "Data".washing.cipRegim, in2 := 3)
      Contact( "Di_1Ga01" )
      Contact( "Di_Ga1.2" )
      I_Contact( "Di_Ga2.2" )
   END_RUNG wire#w1
   RUNG wire#powerrail
      { S7_Templates := "SrcType := Int" } EQ_Contact(in1 := "Data".washing.cipRegim, in2 := 4)
      Contact( "Di_1Ga02" )
      I_Contact( "Di_Ga1.2" )
      Contact( "Di_Ga2.2" )
   END_RUNG wire#w1
   // the same network as SCL:
   "Data".washing.readyRoute := (("Data".washing.cipRegim = 1) AND NOT "Di_Ga1.1" AND NOT "Di_Ga2.1") OR (("Data".washing.cipRegim = 2) AND "Di_1Ga06" AND NOT "Di_Ga1.2" AND NOT "Di_Ga2.2") OR (("Data".washing.cipRegim = 3) AND "Di_1Ga01" AND "Di_Ga1.2" AND NOT "Di_Ga2.2") OR (("Data".washing.cipRegim = 4) AND "Di_1Ga02" AND NOT "Di_Ga1.2" AND "Di_Ga2.2");
END_REGION

REGION Network 2: Разрешение работы
   RUNG wire#powerrail
      { S7_Templates := "SrcType := Int" } EQ_Contact(in1 := "Data".washing.cipRegim, in2 := 1)
      { S7_Templates := "SrcType := Int" } NE_Contact(in1 := "Kr_1_Work"."Step", in2 := 1)
      { S7_Templates := "SrcType := Int" } NE_Contact(in1 := "Kr_2_Work"."Step", in2 := 1)
      wire#w1
      Coil( "Data".ReadyCIP )
   END_RUNG
   RUNG wire#powerrail
      { S7_Templates := "SrcType := Int" } EQ_Contact(in1 := "Data".washing.cipRegim, in2 := 2)
      { S7_Templates := "SrcType := Int" } NE_Contact(in1 := "Kr_1_Work"."Step", in2 := 3)
      { S7_Templates := "SrcType := Int" } NE_Contact(in1 := "Kr_2_Work"."Step", in2 := 3)
   END_RUNG wire#w1
   RUNG wire#powerrail
      { S7_Templates := "SrcType := Int" } EQ_Contact(in1 := "Data".washing.cipRegim, in2 := 3)
      I_Contact( "Kr_1_Work".Run )
      { S7_Templates := "SrcType := Int" } NE_Contact(in1 := "Kr_2_Work"."Step", in2 := 3)
   END_RUNG wire#w1
   RUNG wire#powerrail
      { S7_Templates := "SrcType := Int" } EQ_Contact(in1 := "Data".washing.cipRegim, in2 := 4)
      I_Contact( "Kr_2_Work".Run )
      { S7_Templates := "SrcType := Int" } NE_Contact(in1 := "Kr_1_Work"."Step", in2 := 3)
   END_RUNG wire#w1
   RUNG wire#powerrail
      I_Contact( "Data".EnableReady )
   END_RUNG wire#w1
   // the same network as SCL:
   "Data".ReadyCIP := (("Data".washing.cipRegim = 1) AND ("Kr_1_Work"."Step" <> 1) AND ("Kr_2_Work"."Step" <> 1)) OR (("Data".washing.cipRegim = 2) AND ("Kr_1_Work"."Step" <> 3) AND ("Kr_2_Work"."Step" <> 3)) OR (("Data".washing.cipRegim = 3) AND NOT "Kr_1_Work".Run AND ("Kr_2_Work"."Step" <> 3)) OR (("Data".washing.cipRegim = 4) AND NOT "Kr_2_Work".Run AND ("Kr_1_Work"."Step" <> 3)) OR NOT "Data".EnableReady;
END_REGION

REGION Network 3: Готовность к включению мойки
   RUNG wire#powerrail
      Contact( "Data".washing.readyRoute )
      I_Contact( "Data".GlobalErrorStop )
      I_Contact( "Data".MAN_ON )
      Contact( "Data".ReadyCIP )
      Coil( "Data".washing.readyGlobal )
   END_RUNG
   // the same network as SCL:
   "Data".washing.readyGlobal := "Data".washing.readyRoute AND NOT "Data".GlobalErrorStop AND NOT "Data".MAN_ON AND "Data".ReadyCIP;
END_REGION

REGION Network 4: Таймер на включение
   "IEC_Timer_0_DB".TON(IN := "Data".washing.Start AND "Data".washing.readyGlobal, PT := T#1s);
   "WashingWork_DB".Start := "IEC_Timer_0_DB".Q;
END_REGION

REGION Network 5: Таймер на выключение
   "IEC_Timer_0_DB_1".TON(IN := "Data".washing.Stop, PT := T#1s);
   "WashingWork_DB".Stop := "IEC_Timer_0_DB_1".Q;
END_REGION

REGION Network 6: Блок управления мойки
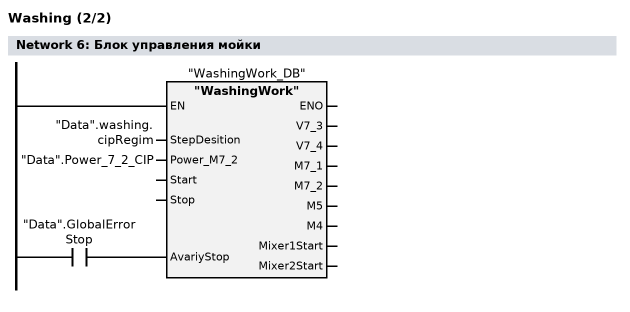
   RUNG wire#powerrail
      "WashingWork_DB"(AvariyStop := wire#w1, StepDesition := "Data".washing.cipRegim, Power_M7_2 := "Data".Power_7_2_CIP, Start :=, Stop :=, V7_3 =>, V7_4 =>, M7_1 =>, M7_2 =>, M5 =>, M4 =>, Mixer1Start =>, Mixer2Start =>)
   END_RUNG
   RUNG wire#powerrail
      Contact( "Data".GlobalErrorStop )
   END_RUNG wire#w1
   // the same network as SCL:
   "WashingWork_DB"(StepDesition := "Data".washing.cipRegim,   // "WashingWork"
                    Power_M7_2 := "Data".Power_7_2_CIP,
                    AvariyStop := "Data".GlobalErrorStop);
END_REGION
END_FUNCTION

// folder: _LIB

